C01805=1100.672,-5.062,-52.510,176.250,14.221,151.801
C01806=1100.666,-5.311,-52.497,176.248,14.221,151.801
C01807=1100.661,-5.561,-52.484,176.246,14.220,151.802
C01808=1100.655,-5.810,-52.470,176.244,14.220,151.802
C01809=1100.649,-6.060,-52.457,176.242,14.219,151.803
C01810=1100.643,-6.309,-52.443,176.240,14.219,151.803
C01811=1100.637,-6.559,-52.429,176.238,14.218,151.803
C01812=1100.631,-6.808,-52.416,176.236,14.218,151.804
C01813=1100.626,-7.058,-52.403,176.234,14.218,151.804
C01814=1100.620,-7.307,-52.390,176.232,14.217,151.804
C01815=1100.614,-7.557,-52.376,176.230,14.216,151.805
C01816=1100.608,-7.806,-52.363,176.228,14.216,151.805
C01817=1100.602,-8.055,-52.349,176.225,14.215,151.805
C01818=1100.597,-8.306,-52.336,176.223,14.214,151.806
C01819=1100.590,-8.555,-52.323,176.221,14.214,151.806
C01820=1100.585,-8.804,-52.309,176.219,14.213,151.807
C01821=1100.578,-9.054,-52.295,176.217,14.213,151.807
C01822=1100.573,-9.305,-52.282,176.215,14.212,151.807
C01823=1100.567,-9.554,-52.269,176.213,14.211,151.808
C01824=1100.561,-9.804,-52.255,176.210,14.211,151.808
C01825=1100.555,-10.053,-52.242,176.208,14.211,151.808
C01826=1100.550,-10.303,-52.229,176.206,14.210,151.809
C01827=1100.544,-10.552,-52.215,176.204,14.210,151.809
C01828=1100.537,-10.801,-52.202,176.202,14.209,151.809
C01829=1100.532,-11.052,-52.189,176.200,14.209,151.810
C01830=1100.526,-11.301,-52.176,176.198,14.208,151.810
C01831=1100.521,-11.551,-52.162,176.195,14.207,151.810
C01832=1100.515,-11.800,-52.149,176.193,14.206,151.811
C01833=1100.509,-12.050,-52.136,176.191,14.206,151.811
C01834=1100.503,-12.299,-52.122,176.189,14.205,151.811
C01835=1100.498,-12.548,-52.110,176.187,14.205,151.812
C01836=1100.492,-12.798,-52.096,176.185,14.204,151.812
C01837=1100.486,-13.047,-52.083,176.183,14.204,151.813
C01838=1100.480,-13.297,-52.070,176.181,14.203,151.813
C01839=1100.475,-13.547,-52.056,176.179,14.203,151.813
C01840=1100.468,-13.796,-52.043,176.177,14.202,151.813
C01841=1100.463,-14.046,-52.030,176.175,14.201,151.814
C01842=1100.457,-14.295,-52.017,176.173,14.201,151.814
C01843=1100.451,-14.545,-52.004,176.171,14.200,151.815
C01844=1100.446,-14.795,-51.990,176.169,14.200,151.815
C01845=1100.440,-15.045,-51.978,176.167,14.199,151.815
C01846=1100.434,-15.294,-51.965,176.165,14.198,151.816
C01847=1100.428,-15.544,-51.951,176.163,14.198,151.816
C01848=1100.422,-15.794,-51.938,176.160,14.197,151.816
C01849=1100.416,-16.061,-51.924,176.158,14.196,151.817
C01850=1100.409,-16.328,-51.910,176.156,14.196,151.817
C01851=1100.403,-16.596,-51.896,176.154,14.195,151.817
C01852=1100.397,-16.863,-51.882,176.152,14.195,151.818
C01853=1100.391,-17.113,-51.869,176.150,14.194,151.818
C01854=1100.385,-17.362,-51.856,176.148,14.194,151.818
C01855=1100.379,-17.612,-51.843,176.145,14.194,151.819
C01856=1100.373,-17.861,-51.830,176.144,14.193,151.819
C01857=1100.367,-18.111,-51.817,176.141,14.193,151.820
C01858=1100.362,-18.360,-51.804,176.140,14.192,151.820
C01859=1100.356,-18.610,-51.791,176.137,14.191,151.820
C01860=1100.350,-18.859,-51.778,176.135,14.190,151.821
C01861=1100.344,-19.109,-51.765,176.133,14.190,151.821
C01862=1100.338,-19.358,-51.752,176.131,14.189,151.821
C01863=1100.333,-19.609,-51.739,176.128,14.189,151.822
C01864=1100.327,-19.858,-51.726,176.127,14.188,151.822
C01865=1100.321,-20.108,-51.713,176.125,14.187,151.822
C01866=1100.315,-20.358,-51.701,176.123,14.187,151.823
C01867=1100.309,-20.607,-51.687,176.121,14.186,151.823
C01868=1100.303,-20.857,-51.675,176.118,14.186,151.823
C01869=1100.298,-21.106,-51.661,176.117,14.185,151.824
C01870=1100.292,-21.356,-51.649,176.114,14.185,151.824
C01871=1100.286,-21.606,-51.636,176.113,14.184,151.824
C01872=1100.280,-21.855,-51.623,176.110,14.184,151.825
C01873=1100.274,-22.105,-51.610,176.108,14.183,151.825
C01874=1100.268,-22.354,-51.597,176.106,14.183,151.825
C01875=1100.262,-22.604,-51.584,176.104,14.182,151.826
C01876=1100.257,-22.853,-51.572,176.102,14.181,151.826
C01877=1100.251,-23.103,-51.558,176.100,14.181,151.826
C01878=1100.245,-23.352,-51.546,176.098,14.180,151.827
C01879=1100.239,-23.602,-51.533,176.096,14.180,151.827
C01880=1100.233,-23.852,-51.520,176.094,14.179,151.827
C01881=1100.227,-24.101,-51.508,176.092,14.178,151.828
C01882=1100.221,-24.351,-51.495,176.090,14.178,151.828
C01883=1100.215,-24.600,-51.482,176.088,14.177,151.828
C01884=1100.210,-24.850,-51.469,176.086,14.177,151.829
C01885=1100.204,-25.100,-51.456,176.084,14.176,151.829
C01886=1100.198,-25.350,-51.444,176.082,14.176,151.829
C01887=1100.192,-25.599,-51.431,176.080,14.175,151.830
C01888=1100.187,-25.848,-51.418,176.078,14.174,151.830
C01889=1100.181,-26.098,-51.406,176.076,14.174,151.830
C01890=1100.175,-26.348,-51.393,176.074,14.173,151.831
C01891=1100.169,-26.597,-51.380,176.072,14.173,151.831
C01892=1100.163,-26.847,-51.367,176.070,14.172,151.831
C01893=1100.158,-27.096,-51.355,176.068,14.172,151.832
C01894=1100.152,-27.346,-51.343,176.066,14.171,151.832
C01895=1100.146,-27.596,-51.329,176.064,14.170,151.832
C01896=1100.140,-27.845,-51.317,176.062,14.170,151.833
C01897=1100.134,-28.095,-51.304,176.060,14.169,151.833
C01898=1100.128,-28.345,-51.292,176.058,14.169,151.833
C01899=1100.123,-28.594,-51.280,176.056,14.168,151.834
C01900=1100.116,-28.844,-51.266,176.054,14.168,151.834
C01901=1100.110,-29.094,-51.254,176.052,14.167,151.834
C01902=1100.105,-29.343,-51.241,176.050,14.166,151.835
C01903=1100.099,-29.593,-51.229,176.048,14.166,151.835
C01904=1100.093,-29.842,-51.216,176.046,14.165,151.835
C01905=1100.087,-30.092,-51.204,176.044,14.165,151.836
C01906=1100.080,-30.341,-51.191,176.042,14.164,151.836
C01907=1100.075,-30.591,-51.179,176.040,14.164,151.836
C01908=1100.069,-30.841,-51.166,176.038,14.163,151.837
C01909=1100.063,-31.090,-51.154,176.036,14.162,151.837
C01910=1100.057,-31.340,-51.141,176.034,14.162,151.837
C01911=1100.052,-31.590,-51.129,176.032,14.161,151.838
C01912=1100.046,-31.840,-51.116,176.030,14.161,151.838
C01913=1100.039,-32.106,-51.104,176.028,14.160,151.838
C01914=1100.033,-32.372,-51.089,176.026,14.160,151.839
C01915=1100.026,-32.639,-51.076,176.024,14.159,151.839
C01916=1100.021,-32.906,-51.063,176.022,14.158,151.839
C01917=1100.015,-33.156,-51.050,176.020,14.158,151.840
C01918=1100.008,-33.405,-51.038,176.018,14.157,151.840
C01919=1100.003,-33.654,-51.026,176.016,14.157,151.840
C01920=1099.997,-33.904,-51.014,176.014,14.156,151.841
C01921=1099.991,-34.154,-51.001,176.012,14.156,151.841
C01922=1099.985,-34.404,-50.989,176.010,14.155,151.841
C01923=1099.980,-34.653,-50.976,176.008,14.154,151.842
C01924=1099.973,-34.903,-50.964,176.006,14.154,151.842
C01925=1099.967,-35.153,-50.952,176.004,14.153,151.842
C01926=1099.962,-35.402,-50.940,176.002,14.153,151.843
C01927=1099.956,-35.652,-50.927,176.000,14.152,151.843
C01928=1099.950,-35.902,-50.915,175.998,14.152,151.843
C01929=1099.944,-36.152,-50.902,175.996,14.151,151.844
C01930=1099.938,-36.400,-50.890,175.994,14.151,151.844
C01931=1099.932,-36.650,-50.878,175.993,14.150,151.844
C01932=1099.927,-36.900,-50.865,175.991,14.150,151.844
C01933=1099.921,-37.149,-50.853,175.989,14.149,151.845
C01934=1099.915,-37.399,-50.841,175.987,14.148,151.845
C01935=1099.909,-37.649,-50.828,175.985,14.148,151.845
C01936=1099.903,-37.898,-50.816,175.983,14.147,151.846
C01937=1099.897,-38.148,-50.804,175.981,14.147,151.846
C01938=1099.892,-38.398,-50.791,175.978,14.146,151.847
C01939=1099.887,-38.648,-50.780,175.977,14.146,151.847
C01940=1099.880,-38.897,-50.768,175.975,14.145,151.847
C01941=1099.874,-39.147,-50.755,175.973,14.144,151.848
C01942=1099.869,-39.396,-50.743,175.971,14.144,151.848
C01943=1099.862,-39.646,-50.731,175.969,14.143,151.848
C01944=1099.856,-39.896,-50.719,175.967,14.143,151.848
C01945=1099.851,-40.145,-50.706,175.965,14.142,151.849
C01946=1099.844,-40.394,-50.694,175.963,14.142,151.849
C01947=1099.838,-40.644,-50.682,175.961,14.141,151.849
C01948=1099.833,-40.894,-50.670,175.959,14.141,151.850
C01949=1099.827,-41.144,-50.658,175.957,14.140,151.850
C01950=1099.821,-41.394,-50.646,175.956,14.140,151.850
C01951=1099.815,-41.643,-50.634,175.953,14.139,151.851
C01952=1099.809,-41.892,-50.622,175.951,14.139,151.851
C01953=1099.803,-42.142,-50.609,175.950,14.138,151.851
C01954=1099.797,-42.392,-50.598,175.947,14.137,151.852
C01955=1099.791,-42.642,-50.586,175.945,14.137,151.852
C01956=1099.785,-42.891,-50.573,175.943,14.136,151.852
C01957=1099.779,-43.140,-50.562,175.941,14.136,151.853
C01958=1099.773,-43.390,-50.549,175.940,14.135,151.853
C01959=1099.768,-43.641,-50.537,175.938,14.135,151.853
C01960=1099.762,-43.890,-50.526,175.936,14.134,151.854
C01961=1099.756,-44.139,-50.513,175.934,14.134,151.854
C01962=1099.750,-44.388,-50.502,175.932,14.133,151.854
C01963=1099.744,-44.639,-50.490,175.930,14.133,151.855
C01964=1099.738,-44.889,-50.477,175.928,14.132,151.855
C01965=1099.732,-45.138,-50.466,175.926,14.131,151.855
C01966=1099.726,-45.387,-50.453,175.924,14.131,151.856
C01967=1099.720,-45.638,-50.442,175.922,14.130,151.856
C01968=1099.715,-45.887,-50.430,175.920,14.130,151.856
C01969=1099.708,-46.136,-50.418,175.919,14.130,151.856
C01970=1099.703,-46.386,-50.406,175.917,14.129,151.857
C01971=1099.697,-46.636,-50.394,175.915,14.128,151.857
C01972=1099.691,-46.885,-50.382,175.913,14.128,151.858
C01973=1099.685,-47.135,-50.370,175.911,14.127,151.858
C01974=1099.679,-47.385,-50.358,175.909,14.127,151.858
C01975=1099.673,-47.634,-50.346,175.907,14.126,151.859
C01976=1099.667,-47.884,-50.335,175.905,14.126,151.859
C01977=1099.661,-48.151,-50.322,175.903,14.125,151.859
C01978=1099.655,-48.419,-50.309,175.901,14.124,151.859
C01979=1099.649,-48.685,-50.296,175.899,14.124,151.860
C01980=1099.643,-48.952,-50.284,175.897,14.123,151.860
C01981=1099.637,-49.202,-50.272,175.895,14.123,151.860
C01982=1099.630,-49.451,-50.260,175.893,14.122,151.861
C01983=1099.625,-49.701,-50.248,175.892,14.122,151.861
C01984=1099.618,-49.951,-50.236,175.890,14.121,151.861
C01985=1099.613,-50.200,-50.225,175.888,14.121,151.862
C01986=1099.607,-50.450,-50.213,175.886,14.120,151.862
C01987=1099.601,-50.699,-50.201,175.884,14.120,151.862
C01988=1099.595,-50.949,-50.189,175.882,14.119,151.863
C01989=1099.589,-51.198,-50.178,175.880,14.119,151.863
C01990=1099.583,-51.449,-50.166,175.878,14.118,151.863
C01991=1099.577,-51.698,-50.154,175.877,14.118,151.864
C01992=1099.571,-51.948,-50.143,175.875,14.117,151.864
C01993=1099.565,-52.198,-50.130,175.873,14.117,151.864
C01994=1099.559,-52.447,-50.119,175.871,14.116,151.865
C01995=1099.553,-52.697,-50.108,175.868,14.116,151.865
C01996=1099.546,-52.946,-50.096,175.867,14.115,151.865
C01997=1099.541,-53.196,-50.084,175.865,14.114,151.866
C01998=1099.534,-53.446,-50.072,175.863,14.115,151.866
C01999=1099.529,-53.695,-50.061,175.861,14.114,151.866
C02000=1099.523,-53.945,-50.049,175.859,14.114,151.867
C02001=1099.517,-54.195,-50.038,175.857,14.113,151.867
C02002=1099.510,-54.444,-50.026,175.855,14.112,151.867
C02003=1099.505,-54.694,-50.015,175.853,14.112,151.868
C02004=1099.499,-54.944,-50.003,175.851,14.111,151.868
C02005=1099.492,-55.194,-49.991,175.850,14.111,151.868
C02006=1099.486,-55.443,-49.980,175.848,14.111,151.869
C02007=1099.481,-55.693,-49.968,175.846,14.110,151.869
C02008=1099.475,-55.942,-49.956,175.844,14.110,151.869
C02009=1099.468,-56.192,-49.945,175.842,14.109,151.870
C02010=1099.462,-56.441,-49.933,175.840,14.109,151.870
C02011=1099.457,-56.692,-49.922,175.839,14.108,151.870
C02012=1099.451,-56.941,-49.911,175.837,14.108,151.870
C02013=1099.444,-57.191,-49.899,175.835,14.107,151.871
C02014=1099.439,-57.440,-49.888,175.833,14.107,151.871
C02015=1099.433,-57.690,-49.875,175.831,14.106,151.872
C02016=1099.427,-57.939,-49.864,175.829,14.106,151.872
C02017=1099.421,-58.190,-49.853,175.828,14.105,151.872
C02018=1099.415,-58.438,-49.842,175.825,14.105,151.872
C02019=1099.408,-58.689,-49.830,175.824,14.104,151.873
C02020=1099.403,-58.938,-49.818,175.821,14.104,151.873
C02021=1099.397,-59.188,-49.807,175.820,14.103,151.873
C02022=1099.391,-59.438,-49.796,175.818,14.103,151.874
C02023=1099.384,-59.687,-49.784,175.816,14.103,151.874
C02024=1099.379,-59.937,-49.773,175.814,14.102,151.874
C02025=1099.373,-60.187,-49.761,175.812,14.102,151.875
C02026=1099.367,-60.436,-49.750,175.810,14.101,151.875
C02027=1099.361,-60.685,-49.739,175.808,14.100,151.875
C02028=1099.355,-60.936,-49.728,175.807,14.101,151.876
C02029=1099.349,-61.185,-49.716,175.805,14.100,151.876
C02030=1099.343,-61.435,-49.704,175.803,14.099,151.876
C02031=1099.337,-61.685,-49.693,175.801,14.099,151.877
C02032=1099.331,-61.934,-49.681,175.799,14.098,151.877
C02033=1099.325,-62.184,-49.671,175.798,14.098,151.877
C02034=1099.319,-62.434,-49.659,175.796,14.098,151.878
C02035=1099.314,-62.684,-49.648,175.794,14.097,151.878
C02036=1099.308,-62.932,-49.636,175.792,14.097,151.878
C02037=1099.301,-63.183,-49.625,175.790,14.096,151.879
C02038=1099.296,-63.432,-49.614,175.788,14.095,151.879
C02039=1099.289,-63.682,-49.603,175.787,14.095,151.879
C02040=1099.283,-63.931,-49.591,175.785,14.095,151.879
C02041=1099.278,-64.200,-49.579,175.783,14.094,151.880
C02042=1099.271,-64.468,-49.567,175.781,14.094,151.880
C02043=1099.264,-64.736,-49.554,175.778,14.093,151.881
C02044=1099.258,-65.005,-49.543,175.777,14.093,151.881
C02045=1099.252,-65.254,-49.532,175.775,14.092,151.881
C02046=1099.246,-65.504,-49.521,175.773,14.092,151.882
C02047=1099.240,-65.754,-49.510,175.771,14.091,151.882
C02048=1099.235,-66.003,-49.498,175.769,14.091,151.882
C02049=1099.228,-66.253,-49.486,175.767,14.090,151.883
C02050=1099.223,-66.503,-49.475,175.765,14.090,151.883
C02051=1099.217,-66.752,-49.465,175.764,14.090,151.883
C02052=1099.210,-67.002,-49.453,175.762,14.089,151.883
C02053=1099.205,-67.252,-49.442,175.760,14.088,151.884
C02054=1099.198,-67.501,-49.430,175.758,14.088,151.884
C02055=1099.192,-67.751,-49.420,175.757,14.088,151.884
C02056=1099.187,-68.000,-49.409,175.755,14.088,151.885
C02057=1099.181,-68.251,-49.397,175.753,14.087,151.885
C02058=1099.175,-68.500,-49.386,175.751,14.086,151.885
C02059=1099.170,-68.750,-49.375,175.749,14.086,151.886
C02060=1099.163,-69.000,-49.364,175.748,14.086,151.886
C02061=1099.157,-69.250,-49.353,175.746,14.085,151.886
C02062=1099.152,-69.499,-49.342,175.744,14.085,151.887
C02063=1099.145,-69.749,-49.330,175.742,14.084,151.887
C02064=1099.139,-69.998,-49.319,175.741,14.084,151.887
C02065=1099.134,-70.248,-49.308,175.738,14.083,151.888
C02066=1099.128,-70.497,-49.298,175.737,14.083,151.888
C02067=1099.121,-70.747,-49.286,175.734,14.082,151.888
C02068=1099.116,-70.997,-49.275,175.733,14.082,151.889
C02069=1099.110,-71.246,-49.265,175.731,14.081,151.889
C02070=1099.104,-71.496,-49.253,175.729,14.081,151.889
C02071=1099.098,-71.746,-49.242,175.727,14.080,151.889
C02072=1099.093,-71.996,-49.231,175.725,14.080,151.890
C02073=1099.087,-72.245,-49.220,175.724,14.080,151.890
C02074=1099.081,-72.495,-49.209,175.722,14.079,151.890
C02075=1099.075,-72.745,-49.198,175.720,14.078,151.891
C02076=1099.069,-72.994,-49.187,175.718,14.078,151.891
C02077=1099.063,-73.245,-49.176,175.717,14.078,151.891
C02078=1099.057,-73.494,-49.165,175.715,14.077,151.892
C02079=1099.052,-73.744,-49.154,175.713,14.077,151.892
C02080=1099.046,-73.993,-49.143,175.711,14.076,151.892
C02081=1099.039,-74.243,-49.132,175.710,14.077,151.893
C02082=1099.034,-74.493,-49.121,175.708,14.076,151.893
C02083=1099.028,-74.742,-49.110,175.706,14.075,151.893
C02084=1099.022,-74.991,-49.100,175.704,14.075,151.894
C02085=1099.015,-75.242,-49.089,175.703,14.075,151.894
C02086=1099.009,-75.491,-49.078,175.700,14.074,151.894
C02087=1099.004,-75.741,-49.067,175.698,14.074,151.895
C02088=1098.997,-75.991,-49.056,175.697,14.074,151.895
C02089=1098.992,-76.240,-49.045,175.695,14.073,151.895
C02090=1098.986,-76.490,-49.034,175.693,14.072,151.896
C02091=1098.979,-76.740,-49.023,175.691,14.072,151.896
C02092=1098.973,-76.990,-49.013,175.690,14.072,151.896
C02093=1098.968,-77.239,-49.002,175.688,14.072,151.897
C02094=1098.962,-77.489,-48.991,175.686,14.071,151.897
C02095=1098.956,-77.739,-48.980,175.685,14.071,151.897
C02096=1098.950,-77.988,-48.969,175.683,14.071,151.898
C02097=1098.943,-78.238,-48.959,175.681,14.070,151.898
C02098=1098.938,-78.487,-48.948,175.678,14.070,151.898
C02099=1098.931,-78.737,-48.937,175.677,14.069,151.898
C02100=1098.926,-78.987,-48.926,175.675,14.069,151.899
C02101=1098.920,-79.237,-48.916,175.673,14.068,151.899
C02102=1098.914,-79.486,-48.905,175.672,14.068,151.899
C02103=1098.907,-79.736,-48.894,175.670,14.068,151.900
C02104=1098.902,-79.986,-48.883,175.668,14.067,151.900
C02105=1098.895,-80.256,-48.871,175.666,14.067,151.901
C02106=1098.889,-80.527,-48.860,175.664,14.066,151.901
C02107=1098.882,-80.797,-48.849,175.663,14.066,151.901
C02108=1098.875,-81.068,-48.837,175.660,14.066,151.902
C02109=1098.870,-81.318,-48.826,175.658,14.065,151.902
C02110=1098.863,-81.567,-48.816,175.656,14.065,151.902
C02111=1098.857,-81.817,-48.805,175.655,14.065,151.903
C02112=1098.851,-82.066,-48.794,175.653,14.065,151.903
C02113=1098.845,-82.316,-48.784,175.651,14.064,151.903
C02114=1098.839,-82.566,-48.773,175.650,14.064,151.904
C02115=1098.832,-82.816,-48.763,175.648,14.064,151.904
C02116=1098.826,-83.065,-48.752,175.646,14.063,151.904
C02117=1098.821,-83.315,-48.742,175.644,14.063,151.905
C02118=1098.814,-83.564,-48.731,175.643,14.062,151.905
C02119=1098.808,-83.815,-48.720,175.640,14.062,151.905
C02120=1098.802,-84.064,-48.709,175.639,14.062,151.906
C02121=1098.796,-84.314,-48.700,175.637,14.062,151.906
C02122=1098.790,-84.563,-48.689,175.635,14.061,151.906
C02123=1098.784,-84.814,-48.678,175.634,14.061,151.907
C02124=1098.778,-85.063,-48.667,175.632,14.061,151.907
C02125=1098.772,-85.313,-48.657,175.630,14.060,151.907
C02126=1098.766,-85.562,-48.647,175.629,14.060,151.908
C02127=1098.760,-85.811,-48.636,175.626,14.060,151.908
C02128=1098.754,-86.062,-48.625,175.625,14.059,151.908
C02129=1098.748,-86.311,-48.615,175.623,14.059,151.909
C02130=1098.742,-86.561,-48.604,175.621,14.059,151.909
C02131=1098.735,-86.810,-48.594,175.619,14.058,151.909
C02132=1098.730,-87.060,-48.584,175.618,14.058,151.910
C02133=1098.724,-87.310,-48.573,175.616,14.058,151.910
C02134=1098.717,-87.560,-48.562,175.614,14.057,151.910
C02135=1098.712,-87.810,-48.552,175.612,14.058,151.911
C02136=1098.705,-88.059,-48.542,175.610,14.057,151.911
C02137=1098.699,-88.308,-48.531,175.608,14.057,151.911
C02138=1098.693,-88.559,-48.520,175.607,14.056,151.912
C02139=1098.687,-88.808,-48.510,175.605,14.056,151.912
C02140=1098.681,-89.058,-48.500,175.603,14.055,151.912
C02141=1098.675,-89.308,-48.490,175.602,14.056,151.913
C02142=1098.669,-89.557,-48.479,175.600,14.055,151.913
C02143=1098.663,-89.807,-48.469,175.598,14.055,151.913
C02144=1098.657,-90.056,-48.458,175.596,14.055,151.914
C02145=1098.651,-90.307,-48.448,175.594,14.054,151.914
C02146=1098.645,-90.556,-48.438,175.593,14.054,151.914
C02147=1098.639,-90.806,-48.427,175.591,14.054,151.915
C02148=1098.633,-91.056,-48.417,175.589,14.053,151.915
C02149=1098.627,-91.305,-48.406,175.588,14.053,151.915
C02150=1098.621,-91.555,-48.397,175.586,14.053,151.916
C02151=1098.615,-91.804,-48.386,175.584,14.052,151.916
C02152=1098.608,-92.055,-48.376,175.582,14.052,151.916
C02153=1098.603,-92.304,-48.365,175.580,14.052,151.917
C02154=1098.596,-92.554,-48.355,175.578,14.051,151.917
C02155=1098.591,-92.804,-48.345,175.577,14.052,151.917
C02156=1098.584,-93.053,-48.334,175.575,14.051,151.918
C02157=1098.579,-93.303,-48.324,175.574,14.051,151.918
C02158=1098.573,-93.553,-48.313,175.572,14.050,151.918
C02159=1098.567,-93.802,-48.304,175.570,14.050,151.919
C02160=1098.561,-94.052,-48.293,175.568,14.050,151.919
C02161=1098.554,-94.302,-48.283,175.566,14.050,151.919
C02162=1098.549,-94.552,-48.272,175.564,14.049,151.920
C02163=1098.543,-94.802,-48.262,175.563,14.049,151.920
C02164=1098.537,-95.051,-48.252,175.561,14.049,151.920
C02165=1098.531,-95.301,-48.242,175.560,14.049,151.921
C02166=1098.525,-95.550,-48.231,175.558,14.048,151.921
C02167=1098.519,-95.800,-48.222,175.555,14.048,151.921
C02168=1098.513,-96.050,-48.211,175.554,14.048,151.922
C02169=1098.506,-96.323,-48.201,175.552,14.048,151.922
C02170=1098.500,-96.595,-48.189,175.550,14.047,151.922
C02171=1098.493,-96.868,-48.178,175.549,14.047,151.923
C02172=1098.486,-97.141,-48.167,175.547,14.047,151.923
C02173=1098.481,-97.391,-48.156,175.545,14.046,151.923
C02174=1098.474,-97.640,-48.146,175.543,14.046,151.924
C02175=1098.469,-97.890,-48.136,175.541,14.046,151.924
C02176=1098.463,-98.140,-48.126,175.539,14.045,151.925
C02177=1098.456,-98.389,-48.116,175.538,14.045,151.925
C02178=1098.451,-98.640,-48.106,175.536,14.045,151.925
C02179=1098.444,-98.889,-48.096,175.535,14.045,151.926
C02180=1098.438,-99.138,-48.086,175.533,14.045,151.926
C02181=1098.433,-99.389,-48.076,175.530,14.044,151.926
C02182=1098.426,-99.638,-48.066,175.529,14.044,151.927
C02183=1098.420,-99.888,-48.056,175.527,14.044,151.927
C02184=1098.413,-100.137,-48.045,175.526,14.044,151.927
C02185=1098.408,-100.388,-48.035,175.524,14.044,151.928
C02186=1098.401,-100.637,-48.026,175.522,14.044,151.928
C02187=1098.395,-100.887,-48.015,175.520,14.043,151.928
C02188=1098.389,-101.137,-48.005,175.518,14.043,151.929
C02189=1098.383,-101.386,-47.996,175.517,14.043,151.929
C02190=1098.377,-101.636,-47.985,175.515,14.042,151.929
C02191=1098.371,-101.886,-47.975,175.514,14.043,151.930
C02192=1098.365,-102.136,-47.966,175.512,14.042,151.930
C02193=1098.359,-102.385,-47.955,175.510,14.042,151.931
C02194=1098.353,-102.634,-47.946,175.508,14.042,151.931
C02195=1098.347,-102.885,-47.936,175.506,14.041,151.931
C02196=1098.341,-103.134,-47.925,175.505,14.041,151.931
C02197=1098.334,-103.384,-47.916,175.503,14.041,151.932
C02198=1098.329,-103.634,-47.906,175.501,14.041,151.932
C02199=1098.323,-103.883,-47.896,175.499,14.041,151.933
C02200=1098.316,-104.133,-47.886,175.498,14.041,151.933
C02201=1098.310,-104.382,-47.876,175.496,14.040,151.933
C02202=1098.305,-104.633,-47.866,175.495,14.041,151.934
C02203=1098.298,-104.882,-47.856,175.493,14.040,151.934
C02204=1098.292,-105.132,-47.846,175.491,14.040,151.934
C02205=1098.286,-105.381,-47.837,175.489,14.040,151.935
C02206=1098.280,-105.631,-47.827,175.487,14.039,151.935
C02207=1098.274,-105.881,-47.816,175.486,14.039,151.935
C02208=1098.268,-106.130,-47.807,175.484,14.039,151.936
C02209=1098.262,-106.380,-47.797,175.483,14.039,151.936
C02210=1098.256,-106.630,-47.788,175.480,14.039,151.936
C02211=1098.250,-106.880,-47.777,175.479,14.039,151.937
C02212=1098.244,-107.129,-47.767,175.477,14.038,151.937
C02213=1098.237,-107.379,-47.758,175.476,14.039,151.938
C02214=1098.231,-107.629,-47.748,175.474,14.038,151.938
C02215=1098.225,-107.879,-47.738,175.472,14.038,151.938
C02216=1098.219,-108.129,-47.729,175.470,14.038,151.939
C02217=1098.213,-108.378,-47.718,175.468,14.037,151.939
C02218=1098.207,-108.628,-47.708,175.467,14.038,151.939
C02219=1098.201,-108.878,-47.699,175.465,14.037,151.940
C02220=1098.195,-109.127,-47.689,175.463,14.037,151.940
C02221=1098.189,-109.377,-47.680,175.461,14.037,151.940
C02222=1098.182,-109.627,-47.670,175.460,14.037,151.941
C02223=1098.176,-109.876,-47.660,175.458,14.037,151.941
C02224=1098.170,-110.126,-47.650,175.456,14.037,151.941
C02225=1098.164,-110.376,-47.641,175.455,14.036,151.942
C02226=1098.158,-110.626,-47.631,175.453,14.037,151.942
C02227=1098.152,-110.876,-47.621,175.451,14.036,151.943
C02228=1098.146,-111.125,-47.611,175.450,14.036,151.943
C02229=1098.140,-111.375,-47.602,175.448,14.036,151.943
C02230=1098.133,-111.624,-47.592,175.446,14.036,151.944
C02231=1098.127,-111.874,-47.582,175.444,14.036,151.944
C02232=1098.121,-112.124,-47.572,175.443,14.036,151.944
C02233=1098.115,-112.363,-47.563,175.441,14.036,151.945
C02234=1098.109,-112.602,-47.554,175.440,14.036,151.945
C02235=1098.103,-112.841,-47.545,175.437,14.035,151.945
C02236=1098.098,-113.081,-47.536,175.436,14.036,151.946
C02237=1098.091,-113.319,-47.526,175.434,14.035,151.946
C02238=1098.085,-113.559,-47.517,175.433,14.035,151.946
C02239=1098.080,-113.798,-47.507,175.431,14.035,151.947
C02240=1098.073,-114.037,-47.499,175.429,14.035,151.947
C02241=1098.067,-114.287,-47.489,175.428,14.035,151.948
C02242=1098.062,-114.536,-47.480,175.426,14.034,151.948
C02243=1098.056,-114.786,-47.470,175.425,14.035,151.948
C02244=1098.049,-115.036,-47.461,175.422,14.035,151.949
C02245=1098.043,-115.285,-47.451,175.421,14.034,151.949
C02246=1098.037,-115.535,-47.442,175.419,14.034,151.949
C02247=1098.031,-115.785,-47.432,175.418,14.035,151.950
C02248=1098.025,-116.035,-47.422,175.415,14.034,151.950
C02249=1098.019,-116.285,-47.413,175.414,14.034,151.950
C02250=1098.012,-116.534,-47.403,175.412,14.034,151.951
C02251=1098.006,-116.784,-47.394,175.411,14.034,151.951
C02252=1098.000,-117.034,-47.384,175.409,14.033,151.951
C02253=1097.994,-117.284,-47.375,175.407,14.034,151.952
C02254=1097.988,-117.534,-47.365,175.405,14.034,151.952
C02255=1097.981,-117.783,-47.355,175.404,14.034,151.953
C02256=1097.975,-118.033,-47.346,175.402,14.033,151.953
C02257=1097.970,-118.282,-47.337,175.400,14.034,151.953
C02258=1097.964,-118.532,-47.327,175.398,14.033,151.954
C02259=1097.957,-118.782,-47.318,175.397,14.033,151.954
C02260=1097.951,-119.032,-47.308,175.395,14.033,151.954
C02261=1097.945,-119.281,-47.298,175.393,14.033,151.955
C02262=1097.939,-119.531,-47.289,175.392,14.034,151.955
C02263=1097.933,-119.781,-47.279,175.390,14.033,151.956
C02264=1097.926,-120.030,-47.270,175.389,14.033,151.956
C02265=1097.920,-120.280,-47.261,175.386,14.033,151.956
C02266=1097.914,-120.531,-47.252,175.385,14.033,151.957
C02267=1097.908,-120.781,-47.242,175.383,14.033,151.957
C02268=1097.902,-121.030,-47.233,175.382,14.033,151.957
C02269=1097.896,-121.279,-47.224,175.379,14.033,151.958
C02270=1097.890,-121.529,-47.214,175.378,14.033,151.958
C02271=1097.884,-121.779,-47.204,175.376,14.032,151.959
C02272=1097.877,-122.029,-47.195,175.375,14.033,151.959
C02273=1097.870,-122.278,-47.186,175.373,14.033,151.959
C02274=1097.864,-122.528,-47.176,175.371,14.033,151.960
C02275=1097.858,-122.778,-47.167,175.370,14.033,151.960
C02276=1097.853,-123.028,-47.158,175.368,14.032,151.960
C02277=1097.847,-123.277,-47.149,175.366,14.033,151.961
C02278=1097.840,-123.527,-47.139,175.364,14.032,151.961
C02279=1097.834,-123.777,-47.130,175.363,14.033,151.962
C02280=1097.827,-124.026,-47.121,175.361,14.032,151.962
C02281=1097.821,-124.276,-47.111,175.359,14.032,151.962
C02282=1097.815,-124.527,-47.102,175.358,14.033,151.963
C02283=1097.810,-124.776,-47.093,175.356,14.033,151.963
C02284=1097.804,-125.026,-47.083,175.354,14.032,151.963
C02285=1097.797,-125.275,-47.074,175.352,14.032,151.964
C02286=1097.791,-125.525,-47.065,175.351,14.033,151.964
C02287=1097.784,-125.775,-47.055,175.349,14.032,151.965
C02288=1097.779,-126.025,-47.046,175.347,14.033,151.965
C02289=1097.772,-126.275,-47.037,175.346,14.033,151.965
C02290=1097.765,-126.524,-47.028,175.344,14.032,151.966
C02291=1097.760,-126.773,-47.019,175.342,14.033,151.966
C02292=1097.754,-127.024,-47.010,175.340,14.032,151.967
C02293=1097.746,-127.319,-46.999,175.339,14.033,151.967
C02294=1097.739,-127.615,-46.987,175.337,14.032,151.967
C02295=1097.731,-127.911,-46.977,175.334,14.032,151.968
C02296=1097.726,-128.206,-46.966,175.333,14.033,151.968
C02297=1097.317,-128.228,-47.072,175.291,14.129,151.996
C02298=1097.321,-127.958,-47.082,175.293,14.130,151.996
C02299=1097.328,-127.689,-47.092,175.295,14.129,151.996
C02300=1097.335,-127.419,-47.102,175.297,14.130,151.995
C02301=1097.341,-127.150,-47.112,175.298,14.129,151.995
C02302=1097.347,-126.900,-47.121,175.300,14.130,151.995
C02303=1097.353,-126.650,-47.130,175.302,14.130,151.994
C02304=1097.359,-126.400,-47.140,175.304,14.130,151.994
C02305=1097.366,-126.151,-47.149,175.305,14.129,151.993
C02306=1097.372,-125.901,-47.158,175.307,14.129,151.993
C02307=1097.378,-125.652,-47.167,175.308,14.130,151.993
C02308=1097.384,-125.401,-47.176,175.310,14.129,151.992
C02309=1097.391,-125.152,-47.185,175.312,14.130,151.992
C02310=1097.397,-124.902,-47.195,175.314,14.129,151.991
C02311=1097.403,-124.652,-47.204,175.315,14.130,151.991
C02312=1097.409,-124.402,-47.214,175.317,14.130,151.991
C02313=1097.415,-124.152,-47.223,175.318,14.129,151.990
C02314=1097.421,-123.903,-47.231,175.321,14.130,151.990
C02315=1097.427,-123.653,-47.241,175.322,14.130,151.990
C02316=1097.434,-123.404,-47.250,175.324,14.130,151.989
C02317=1097.440,-123.154,-47.260,175.325,14.130,151.989
C02318=1097.446,-122.904,-47.270,175.327,14.130,151.989
C02319=1097.452,-122.654,-47.279,175.329,14.130,151.988
C02320=1097.458,-122.404,-47.288,175.331,14.130,151.988
C02321=1097.464,-122.155,-47.297,175.332,14.130,151.987
C02322=1097.470,-121.905,-47.306,175.334,14.131,151.987
C02323=1097.477,-121.655,-47.316,175.336,14.130,151.987
C02324=1097.483,-121.406,-47.325,175.337,14.130,151.986
C02325=1097.489,-121.156,-47.335,175.339,14.131,151.986
C02326=1097.495,-120.906,-47.344,175.340,14.130,151.986
C02327=1097.501,-120.656,-47.354,175.343,14.130,151.985
C02328=1097.508,-120.406,-47.364,175.344,14.130,151.985
C02329=1097.513,-120.156,-47.372,175.346,14.131,151.984
C02330=1097.520,-119.907,-47.381,175.347,14.131,151.984
C02331=1097.526,-119.657,-47.391,175.350,14.131,151.984
C02332=1097.532,-119.408,-47.400,175.351,14.131,151.983
C02333=1097.538,-119.158,-47.410,175.353,14.131,151.983
C02334=1097.544,-118.908,-47.419,175.354,14.131,151.983
C02335=1097.551,-118.658,-47.429,175.356,14.132,151.982
C02336=1097.557,-118.408,-47.438,175.358,14.131,151.982
C02337=1097.563,-118.159,-47.448,175.360,14.131,151.981
C02338=1097.569,-117.909,-47.458,175.361,14.132,151.981
C02339=1097.575,-117.659,-47.467,175.363,14.132,151.981
C02340=1097.581,-117.409,-47.477,175.365,14.131,151.980
C02341=1097.587,-117.160,-47.486,175.366,14.132,151.980
C02342=1097.593,-116.910,-47.496,175.368,14.132,151.980
C02343=1097.599,-116.661,-47.505,175.370,14.132,151.979
C02344=1097.605,-116.411,-47.515,175.371,14.132,151.979
C02345=1097.612,-116.161,-47.524,175.373,14.132,151.979
C02346=1097.618,-115.911,-47.534,175.375,14.132,151.978
C02347=1097.624,-115.661,-47.543,175.377,14.133,151.978
C02348=1097.630,-115.412,-47.553,175.378,14.132,151.978
C02349=1097.636,-115.162,-47.562,175.380,14.133,151.977
C02350=1097.643,-114.912,-47.572,175.382,14.133,151.977
C02351=1097.649,-114.662,-47.582,175.384,14.133,151.977
C02352=1097.655,-114.412,-47.591,175.385,14.133,151.976
C02353=1097.661,-114.163,-47.601,175.387,14.133,151.976
C02354=1097.667,-113.913,-47.610,175.388,14.133,151.975
C02355=1097.673,-113.663,-47.620,175.391,14.133,151.975
C02356=1097.679,-113.414,-47.629,175.392,14.133,151.975
C02357=1097.685,-113.164,-47.639,175.394,14.134,151.974
C02358=1097.691,-112.909,-47.649,175.395,14.133,151.974
C02359=1097.698,-112.654,-47.658,175.397,14.134,151.974
C02360=1097.704,-112.399,-47.668,175.399,14.134,151.973
C02361=1097.710,-112.145,-47.678,175.401,14.135,151.973
C02362=1097.716,-111.895,-47.688,175.402,14.134,151.973
C02363=1097.723,-111.646,-47.698,175.404,14.134,151.972
C02364=1097.729,-111.396,-47.707,175.405,14.135,151.972
C02365=1097.735,-111.146,-47.717,175.408,14.135,151.972
C02366=1097.741,-110.896,-47.727,175.409,14.134,151.971
C02367=1097.747,-110.646,-47.736,175.411,14.135,151.971
C02368=1097.753,-110.397,-47.746,175.412,14.135,151.970
C02369=1097.760,-110.147,-47.755,175.414,14.136,151.970
C02370=1097.765,-109.897,-47.766,175.416,14.135,151.970
C02371=1097.772,-109.647,-47.776,175.418,14.135,151.969
C02372=1097.778,-109.398,-47.785,175.420,14.136,151.969
C02373=1097.784,-109.148,-47.795,175.421,14.136,151.969
C02374=1097.790,-108.898,-47.804,175.423,14.137,151.968
C02375=1097.796,-108.648,-47.814,175.425,14.136,151.968
C02376=1097.803,-108.399,-47.824,175.427,14.136,151.968
C02377=1097.809,-108.149,-47.834,175.428,14.137,151.967
C02378=1097.815,-107.900,-47.843,175.430,14.137,151.967
C02379=1097.820,-107.649,-47.854,175.431,14.137,151.967
C02380=1097.827,-107.400,-47.863,175.433,14.137,151.966
C02381=1097.833,-107.150,-47.873,175.435,14.137,151.966
C02382=1097.839,-106.901,-47.883,175.437,14.138,151.966
C02383=1097.845,-106.651,-47.893,175.438,14.137,151.965
C02384=1097.851,-106.401,-47.903,175.440,14.138,151.965
C02385=1097.857,-106.151,-47.912,175.442,14.138,151.965
C02386=1097.864,-105.902,-47.923,175.443,14.138,151.964
C02387=1097.870,-105.652,-47.932,175.446,14.139,151.964
C02388=1097.876,-105.402,-47.942,175.447,14.139,151.964
C02389=1097.881,-105.152,-47.952,175.449,14.139,151.963
C02390=1097.888,-104.903,-47.962,175.450,14.139,151.963
C02391=1097.894,-104.653,-47.972,175.452,14.139,151.963
C02392=1097.900,-104.403,-47.981,175.454,14.139,151.962
C02393=1097.906,-104.153,-47.991,175.455,14.140,151.962
C02394=1097.912,-103.904,-48.002,175.458,14.140,151.961
C02395=1097.918,-103.654,-48.011,175.459,14.140,151.961
C02396=1097.924,-103.404,-48.021,175.461,14.140,151.961
C02397=1097.930,-103.154,-48.031,175.462,14.141,151.961
C02398=1097.936,-102.905,-48.041,175.464,14.141,151.960
C02399=1097.942,-102.655,-48.051,175.465,14.141,151.960
C02400=1097.949,-102.404,-48.061,175.468,14.141,151.959
C02401=1097.955,-102.155,-48.072,175.470,14.142,151.959
C02402=1097.961,-101.906,-48.081,175.471,14.142,151.959
C02403=1097.967,-101.656,-48.091,175.473,14.142,151.958
C02404=1097.973,-101.406,-48.102,175.474,14.142,151.958
C02405=1097.979,-101.156,-48.111,175.476,14.142,151.958
C02406=1097.985,-100.907,-48.121,175.478,14.143,151.957
C02407=1097.991,-100.657,-48.132,175.480,14.143,151.957
C02408=1097.997,-100.407,-48.141,175.482,14.143,151.957
C02409=1098.003,-100.158,-48.151,175.483,14.143,151.956
C02410=1098.009,-99.908,-48.162,175.485,14.144,151.956
C02411=1098.015,-99.658,-48.171,175.486,14.143,151.956
C02412=1098.022,-99.408,-48.181,175.488,14.144,151.955
C02413=1098.027,-99.159,-48.192,175.490,14.145,151.955
C02414=1098.033,-98.909,-48.201,175.492,14.145,151.955
C02415=1098.041,-98.659,-48.212,175.494,14.145,151.954
C02416=1098.047,-98.409,-48.221,175.495,14.145,151.954
C02417=1098.052,-98.159,-48.232,175.497,14.145,151.954
C02418=1098.059,-97.910,-48.242,175.499,14.146,151.953
C02419=1098.064,-97.660,-48.252,175.500,14.146,151.953
C02420=1098.071,-97.411,-48.262,175.502,14.146,151.953
C02421=1098.077,-97.161,-48.272,175.504,14.146,151.952
C02422=1098.083,-96.889,-48.283,175.506,14.147,151.952
C02423=1098.090,-96.616,-48.294,175.508,14.147,151.952
C02424=1098.096,-96.342,-48.305,175.510,14.147,151.951
C02425=1098.103,-96.069,-48.317,175.512,14.148,151.951
C02426=1098.109,-95.820,-48.328,175.513,14.148,151.951
C02427=1098.115,-95.570,-48.337,175.515,14.148,151.950
C02428=1098.120,-95.320,-48.347,175.517,14.148,151.950
C02429=1098.127,-95.071,-48.358,175.519,14.149,151.950
C02430=1098.132,-94.821,-48.368,175.520,14.150,151.949
C02431=1098.139,-94.572,-48.378,175.522,14.149,151.949
C02432=1098.144,-94.321,-48.388,175.524,14.150,151.949
C02433=1098.151,-94.072,-48.399,175.526,14.150,151.948
C02434=1098.156,-93.821,-48.409,175.527,14.150,151.948
C02435=1098.163,-93.572,-48.419,175.529,14.151,151.948
C02436=1098.168,-93.322,-48.429,175.530,14.151,151.947
C02437=1098.175,-93.073,-48.440,175.533,14.151,151.947
C02438=1098.180,-92.823,-48.450,175.534,14.152,151.947
C02439=1098.187,-92.574,-48.460,175.536,14.152,151.946
C02440=1098.192,-92.324,-48.470,175.538,14.152,151.946
C02441=1098.199,-92.074,-48.481,175.540,14.153,151.946
C02442=1098.204,-91.825,-48.491,175.541,14.153,151.945
C02443=1098.210,-91.574,-48.502,175.543,14.153,151.945
C02444=1098.217,-91.325,-48.512,175.545,14.154,151.945
C02445=1098.222,-91.075,-48.522,175.546,14.154,151.944
C02446=1098.229,-90.826,-48.533,175.548,14.155,151.944
C02447=1098.234,-90.576,-48.543,175.550,14.154,151.944
C02448=1098.241,-90.326,-48.553,175.551,14.155,151.943
C02449=1098.247,-90.077,-48.564,175.554,14.155,151.943
C02450=1098.253,-89.826,-48.574,175.555,14.155,151.943
C02451=1098.259,-89.577,-48.585,175.557,14.156,151.942
C02452=1098.264,-89.327,-48.595,175.559,14.156,151.942
C02453=1098.271,-89.078,-48.605,175.560,14.156,151.942
C02454=1098.277,-88.828,-48.616,175.562,14.157,151.941
C02455=1098.283,-88.578,-48.626,175.564,14.158,151.941
C02456=1098.289,-88.328,-48.637,175.565,14.157,151.941
C02457=1098.296,-88.079,-48.647,175.567,14.158,151.940
C02458=1098.301,-87.829,-48.657,175.570,14.158,151.940
C02459=1098.307,-87.579,-48.668,175.571,14.158,151.940
C02460=1098.313,-87.330,-48.678,175.573,14.159,151.939
C02461=1098.319,-87.080,-48.689,175.575,14.159,151.939
C02462=1098.326,-86.830,-48.699,175.576,14.159,151.939
C02463=1098.331,-86.580,-48.710,175.578,14.160,151.938
C02464=1098.337,-86.331,-48.720,175.580,14.160,151.938
C02465=1098.343,-86.081,-48.731,175.581,14.160,151.938
C02466=1098.350,-85.831,-48.742,175.583,14.161,151.938
C02467=1098.356,-85.581,-48.751,175.585,14.161,151.937
C02468=1098.362,-85.332,-48.762,175.587,14.161,151.937
C02469=1098.367,-85.082,-48.773,175.588,14.162,151.937
C02470=1098.374,-84.833,-48.783,175.591,14.162,151.936
C02471=1098.380,-84.582,-48.794,175.592,14.162,151.936
C02472=1098.386,-84.333,-48.804,175.594,14.163,151.936
C02473=1098.392,-84.084,-48.815,175.596,14.163,151.935
C02474=1098.398,-83.834,-48.825,175.597,14.164,151.935
C02475=1098.405,-83.584,-48.836,175.599,14.164,151.935
C02476=1098.410,-83.334,-48.847,175.601,14.165,151.934
C02477=1098.416,-83.085,-48.858,175.603,14.165,151.934
C02478=1098.422,-82.835,-48.867,175.604,14.165,151.934
C02479=1098.429,-82.585,-48.879,175.607,14.165,151.933
C02480=1098.434,-82.335,-48.889,175.608,14.166,151.933
C02481=1098.441,-82.086,-48.900,175.610,14.166,151.933
C02482=1098.447,-81.837,-48.911,175.612,14.166,151.932
C02483=1098.453,-81.586,-48.921,175.614,14.167,151.932
C02484=1098.459,-81.337,-48.931,175.615,14.167,151.932
C02485=1098.465,-81.087,-48.942,175.617,14.168,151.931
C02486=1098.472,-80.817,-48.954,175.619,14.168,151.931
C02487=1098.478,-80.546,-48.966,175.621,14.169,151.931
C02488=1098.485,-80.275,-48.977,175.623,14.169,151.930
C02489=1098.491,-80.005,-48.989,175.625,14.170,151.930
C02490=1098.497,-79.755,-49.000,175.627,14.169,151.930
C02491=1098.504,-79.505,-49.010,175.628,14.170,151.929
C02492=1098.510,-79.256,-49.021,175.630,14.171,151.929
C02493=1098.515,-79.006,-49.031,175.632,14.170,151.929
C02494=1098.521,-78.756,-49.042,175.634,14.171,151.928
C02495=1098.527,-78.506,-49.053,175.635,14.172,151.928
C02496=1098.534,-78.257,-49.064,175.638,14.172,151.928
C02497=1098.539,-78.008,-49.074,175.639,14.172,151.927
C02498=1098.546,-77.757,-49.086,175.641,14.173,151.927
C02499=1098.551,-77.508,-49.097,175.643,14.173,151.927
C02500=1098.557,-77.258,-49.107,175.644,14.174,151.927
C02501=1098.563,-77.008,-49.118,175.646,14.174,151.926
C02502=1098.570,-76.758,-49.128,175.648,14.175,151.926
C02503=1098.575,-76.509,-49.139,175.650,14.175,151.926
C02504=1098.581,-76.259,-49.150,175.651,14.175,151.925
C02505=1098.587,-76.009,-49.161,175.653,14.176,151.925
C02506=1098.593,-75.760,-49.172,175.655,14.176,151.925
C02507=1098.599,-75.510,-49.183,175.657,14.177,151.924
C02508=1098.605,-75.260,-49.194,175.658,14.177,151.924
C02509=1098.612,-75.011,-49.205,175.660,14.178,151.924
C02510=1098.617,-74.761,-49.215,175.662,14.178,151.923
C02511=1098.623,-74.512,-49.226,175.664,14.179,151.923
C02512=1098.630,-74.262,-49.238,175.666,14.178,151.923
C02513=1098.635,-74.012,-49.248,175.668,14.179,151.922
C02514=1098.641,-73.763,-49.259,175.670,14.180,151.922
C02515=1098.647,-73.512,-49.271,175.671,14.181,151.922
C02516=1098.653,-73.263,-49.281,175.673,14.180,151.921
C02517=1098.659,-73.014,-49.292,175.675,14.181,151.921
C02518=1098.665,-72.764,-49.303,175.677,14.182,151.921
C02519=1098.671,-72.514,-49.314,175.679,14.182,151.920
C02520=1098.677,-72.264,-49.325,175.680,14.182,151.920
C02521=1098.682,-72.015,-49.336,175.682,14.183,151.920
C02522=1098.688,-71.765,-49.347,175.684,14.183,151.920
C02523=1098.694,-71.515,-49.358,175.686,14.184,151.919
C02524=1098.699,-71.265,-49.370,175.687,14.184,151.919
C02525=1098.705,-71.016,-49.381,175.689,14.185,151.919
C02526=1098.712,-70.766,-49.392,175.691,14.185,151.918
C02527=1098.717,-70.516,-49.403,175.693,14.186,151.918
C02528=1098.723,-70.267,-49.414,175.695,14.187,151.918
C02529=1098.729,-70.017,-49.425,175.696,14.186,151.917
C02530=1098.735,-69.767,-49.436,175.698,14.187,151.917
C02531=1098.741,-69.518,-49.447,175.700,14.188,151.917
C02532=1098.747,-69.268,-49.458,175.702,14.189,151.917
C02533=1098.753,-69.018,-49.469,175.703,14.188,151.916
C02534=1098.759,-68.769,-49.480,175.705,14.189,151.916
C02535=1098.765,-68.520,-49.491,175.707,14.190,151.916
C02536=1098.771,-68.269,-49.502,175.709,14.190,151.915
C02537=1098.776,-68.020,-49.514,175.711,14.191,151.915
C02538=1098.782,-67.770,-49.525,175.712,14.191,151.915
C02539=1098.788,-67.520,-49.536,175.714,14.191,151.914
C02540=1098.794,-67.270,-49.547,175.716,14.192,151.914
C02541=1098.800,-67.021,-49.558,175.718,14.193,151.914
C02542=1098.806,-66.771,-49.570,175.720,14.193,151.914
C02543=1098.812,-66.522,-49.581,175.721,14.193,151.913
C02544=1098.818,-66.272,-49.592,175.723,14.194,151.913
C02545=1098.824,-66.022,-49.603,175.725,14.195,151.913
C02546=1098.830,-65.773,-49.614,175.727,14.195,151.912
C02547=1098.836,-65.523,-49.626,175.729,14.196,151.912
C02548=1098.841,-65.273,-49.637,175.730,14.196,151.912
C02549=1098.847,-65.024,-49.648,175.733,14.196,151.911
C02550=1098.854,-64.755,-49.660,175.734,14.197,151.911
C02551=1098.860,-64.487,-49.672,175.736,14.198,151.911
C02552=1098.866,-64.218,-49.684,175.739,14.198,151.910
C02553=1098.873,-63.950,-49.697,175.740,14.199,151.910
C02554=1098.879,-63.700,-49.708,175.742,14.199,151.910
C02555=1098.885,-63.451,-49.719,175.745,14.200,151.909
C02556=1098.891,-63.200,-49.730,175.746,14.200,151.909
C02557=1098.897,-62.952,-49.741,175.747,14.201,151.909
C02558=1098.903,-62.701,-49.753,175.750,14.201,151.908
C02559=1098.908,-62.452,-49.764,175.752,14.202,151.908
C02560=1098.915,-62.201,-49.775,175.753,14.202,151.908
C02561=1098.921,-61.953,-49.787,175.755,14.202,151.908
C02562=1098.927,-61.703,-49.798,175.757,14.203,151.907
C02563=1098.933,-61.453,-49.809,175.759,14.204,151.907
C02564=1098.938,-61.204,-49.821,175.761,14.204,151.907
C02565=1098.945,-60.953,-49.833,175.763,14.205,151.906
C02566=1098.950,-60.704,-49.843,175.765,14.205,151.906
C02567=1098.957,-60.454,-49.855,175.766,14.206,151.906
C02568=1098.963,-60.205,-49.866,175.768,14.206,151.905
C02569=1098.968,-59.954,-49.878,175.770,14.207,151.905
C02570=1098.974,-59.706,-49.890,175.772,14.207,151.905
C02571=1098.980,-59.456,-49.901,175.774,14.208,151.904
C02572=1098.986,-59.206,-49.912,175.775,14.208,151.904
C02573=1098.992,-58.957,-49.923,175.777,14.209,151.904
C02574=1098.998,-58.707,-49.935,175.779,14.209,151.903
C02575=1099.004,-58.457,-49.946,175.781,14.210,151.903
C02576=1099.010,-58.207,-49.958,175.783,14.210,151.903
C02577=1099.016,-57.958,-49.969,175.785,14.211,151.903
C02578=1099.022,-57.708,-49.982,175.787,14.211,151.902
C02579=1099.028,-57.459,-49.992,175.788,14.211,151.902
C02580=1099.034,-57.208,-50.004,175.790,14.212,151.902
C02581=1099.040,-56.960,-50.015,175.792,14.213,151.901
C02582=1099.046,-56.709,-50.027,175.794,14.213,151.901
C02583=1099.052,-56.460,-50.039,175.796,14.214,151.901
C02584=1099.058,-56.210,-50.050,175.798,14.214,151.900
C02585=1099.064,-55.961,-50.062,175.799,14.214,151.900
C02586=1099.070,-55.711,-50.073,175.801,14.215,151.900
C02587=1099.076,-55.461,-50.085,175.803,14.216,151.899
C02588=1099.082,-55.212,-50.096,175.805,14.216,151.899
C02589=1099.089,-54.961,-50.107,175.807,14.217,151.899
C02590=1099.094,-54.712,-50.120,175.809,14.217,151.899
C02591=1099.100,-54.462,-50.131,175.811,14.218,151.898
C02592=1099.106,-54.213,-50.142,175.812,14.218,151.898
C02593=1099.113,-53.963,-50.154,175.814,14.219,151.898
C02594=1099.118,-53.714,-50.166,175.816,14.219,151.897
C02595=1099.124,-53.464,-50.177,175.818,14.220,151.897
C02596=1099.131,-53.214,-50.189,175.820,14.220,151.897
C02597=1099.136,-52.965,-50.201,175.822,14.221,151.896
C02598=1099.143,-52.715,-50.213,175.824,14.221,151.896
C02599=1099.149,-52.466,-50.224,175.825,14.222,151.896
C02600=1099.155,-52.216,-50.235,175.827,14.222,151.895
C02601=1099.160,-51.966,-50.248,175.829,14.223,151.895
C02602=1099.167,-51.716,-50.259,175.831,14.223,151.895
C02603=1099.173,-51.467,-50.271,175.833,14.224,151.894
C02604=1099.178,-51.217,-50.282,175.835,14.224,151.894
C02605=1099.185,-50.967,-50.294,175.837,14.225,151.894
C02606=1099.191,-50.718,-50.306,175.839,14.226,151.894
C02607=1099.197,-50.468,-50.318,175.841,14.226,151.893
C02608=1099.203,-50.218,-50.330,175.842,14.226,151.893
C02609=1099.208,-49.968,-50.341,175.844,14.227,151.893
C02610=1099.215,-49.719,-50.353,175.847,14.227,151.892
C02611=1099.220,-49.470,-50.365,175.848,14.228,151.892
C02612=1099.226,-49.220,-50.376,175.850,14.229,151.892
C02613=1099.232,-48.970,-50.389,175.852,14.230,151.891
C02614=1099.238,-48.703,-50.401,175.854,14.230,151.891
C02615=1099.245,-48.436,-50.414,175.856,14.231,151.891
C02616=1099.251,-48.169,-50.427,175.858,14.231,151.890
C02617=1099.257,-47.902,-50.439,175.860,14.232,151.890
C02618=1099.263,-47.652,-50.451,175.862,14.233,151.890
C02619=1099.269,-47.403,-50.463,175.864,14.233,151.889
C02620=1099.274,-47.152,-50.475,175.866,14.234,151.889
C02621=1099.281,-46.903,-50.487,175.868,14.234,151.889
C02622=1099.286,-46.654,-50.499,175.869,14.234,151.889
C02623=1099.292,-46.403,-50.510,175.871,14.235,151.888
C02624=1099.298,-46.154,-50.522,175.873,14.236,151.888
C02625=1099.304,-45.905,-50.534,175.875,14.236,151.888
C02626=1099.310,-45.654,-50.546,175.877,14.237,151.887
C02627=1099.316,-45.405,-50.558,175.879,14.237,151.887
C02628=1099.322,-45.155,-50.570,175.881,14.238,151.887
C02629=1099.327,-44.906,-50.583,175.883,14.239,151.886
C02630=1099.334,-44.656,-50.594,175.885,14.239,151.886
C02631=1099.340,-44.406,-50.606,175.887,14.240,151.886
C02632=1099.346,-44.157,-50.618,175.889,14.241,151.885
C02633=1099.351,-43.907,-50.631,175.890,14.241,151.885
C02634=1099.356,-43.658,-50.642,175.892,14.241,151.885
C02635=1099.363,-43.408,-50.654,175.894,14.242,151.885
C02636=1099.369,-43.158,-50.667,175.896,14.243,151.884
C02637=1099.375,-42.909,-50.678,175.898,14.243,151.884
C02638=1099.381,-42.659,-50.691,175.900,14.244,151.884
C02639=1099.387,-42.409,-50.703,175.902,14.244,151.883
C02640=1099.393,-42.160,-50.714,175.904,14.245,151.883
C02641=1099.399,-41.910,-50.727,175.906,14.246,151.883
C02642=1099.404,-41.660,-50.739,175.908,14.246,151.882
C02643=1099.410,-41.411,-50.751,175.910,14.247,151.882
C02644=1099.416,-41.161,-50.763,175.912,14.247,151.882
C02645=1099.423,-40.911,-50.775,175.914,14.248,151.881
C02646=1099.428,-40.662,-50.787,175.915,14.248,151.881
C02647=1099.434,-40.412,-50.799,175.917,14.249,151.881
C02648=1099.441,-40.163,-50.811,175.919,14.249,151.880
C02649=1099.446,-39.913,-50.824,175.921,14.250,151.880
C02650=1099.452,-39.664,-50.836,175.923,14.250,151.880
C02651=1099.458,-39.414,-50.848,175.925,14.251,151.880
C02652=1099.463,-39.164,-50.859,175.927,14.252,151.879
C02653=1099.469,-38.914,-50.872,175.929,14.252,151.879
C02654=1099.476,-38.665,-50.884,175.931,14.253,151.879
C02655=1099.481,-38.416,-50.896,175.933,14.254,151.878
C02656=1099.487,-38.166,-50.909,175.935,14.254,151.878
C02657=1099.493,-37.916,-50.921,175.937,14.255,151.878
C02658=1099.498,-37.667,-50.933,175.939,14.256,151.877
C02659=1099.505,-37.417,-50.945,175.941,14.256,151.877
C02660=1099.511,-37.167,-50.958,175.943,14.257,151.877
C02661=1099.516,-36.918,-50.970,175.945,14.257,151.876
C02662=1099.522,-36.668,-50.983,175.946,14.258,151.876
C02663=1099.528,-36.418,-50.995,175.949,14.258,151.876
C02664=1099.534,-36.169,-51.007,175.951,14.259,151.875
C02665=1099.540,-35.919,-51.019,175.952,14.260,151.875
C02666=1099.546,-35.670,-51.032,175.954,14.260,151.875
C02667=1099.552,-35.419,-51.044,175.956,14.260,151.875
C02668=1099.557,-35.170,-51.056,175.958,14.261,151.874
C02669=1099.563,-34.920,-51.069,175.960,14.261,151.874
C02670=1099.569,-34.670,-51.081,175.962,14.262,151.874
C02671=1099.575,-34.422,-51.093,175.964,14.263,151.873
C02672=1099.581,-34.172,-51.106,175.965,14.264,151.873
C02673=1099.587,-33.922,-51.119,175.968,14.264,151.873
C02674=1099.593,-33.672,-51.131,175.969,14.265,151.872
C02675=1099.598,-33.423,-51.143,175.971,14.266,151.872
C02676=1099.604,-33.173,-51.156,175.974,14.266,151.872
C02677=1099.611,-32.924,-51.168,175.975,14.267,151.871
C02678=1099.616,-32.657,-51.181,175.977,14.267,151.871
C02679=1099.623,-32.390,-51.194,175.979,14.268,151.871
C02680=1099.629,-32.123,-51.208,175.981,14.268,151.870
C02681=1099.636,-31.856,-51.221,175.984,14.269,151.870
C02682=1099.642,-31.607,-51.233,175.986,14.270,151.870
C02683=1099.647,-31.357,-51.246,175.988,14.271,151.869
C02684=1099.653,-31.107,-51.258,175.990,14.271,151.869
C02685=1099.659,-30.858,-51.271,175.992,14.272,151.869
C02686=1099.665,-30.608,-51.284,175.994,14.273,151.869
C02687=1099.671,-30.358,-51.296,175.996,14.273,151.868
C02688=1099.676,-30.109,-51.309,175.997,14.273,151.868
C02689=1099.682,-29.859,-51.321,175.999,14.274,151.868
C02690=1099.688,-29.609,-51.334,176.001,14.274,151.867
C02691=1099.695,-29.360,-51.346,176.003,14.275,151.867
C02692=1099.701,-29.110,-51.358,176.005,14.275,151.867
C02693=1099.706,-28.861,-51.371,176.007,14.276,151.866
C02694=1099.712,-28.612,-51.384,176.009,14.277,151.866
C02695=1099.718,-28.362,-51.396,176.011,14.277,151.866
C02696=1099.724,-28.112,-51.409,176.013,14.278,151.865
C02697=1099.730,-27.862,-51.421,176.015,14.279,151.865
C02698=1099.735,-27.613,-51.434,176.017,14.279,151.865
C02699=1099.741,-27.363,-51.447,176.019,14.280,151.864
C02700=1099.747,-27.114,-51.459,176.021,14.280,151.864
C02701=1099.753,-26.864,-51.472,176.023,14.281,151.864
C02702=1099.759,-26.614,-51.485,176.025,14.282,151.863
C02703=1099.765,-26.365,-51.497,176.027,14.282,151.863
C02704=1099.771,-26.115,-51.510,176.029,14.283,151.863
C02705=1099.776,-25.866,-51.523,176.031,14.283,151.862
C02706=1099.783,-25.616,-51.536,176.033,14.284,151.862
C02707=1099.789,-25.366,-51.548,176.035,14.285,151.862
C02708=1099.793,-25.117,-51.561,176.038,14.286,151.861
C02709=1099.799,-24.867,-51.574,176.040,14.287,151.861
C02710=1099.805,-24.618,-51.587,176.042,14.287,151.861
C02711=1099.811,-24.368,-51.600,176.044,14.288,151.861
C02712=1099.817,-24.118,-51.612,176.046,14.288,151.860
C02713=1099.823,-23.869,-51.625,176.048,14.289,151.860
C02714=1099.829,-23.620,-51.638,176.050,14.290,151.860
C02715=1099.834,-23.370,-51.650,176.052,14.290,151.859
C02716=1099.840,-23.120,-51.663,176.054,14.291,151.859
C02717=1099.846,-22.870,-51.677,176.056,14.291,151.859
C02718=1099.852,-22.620,-51.689,176.058,14.292,151.858
C02719=1099.858,-22.371,-51.702,176.060,14.292,151.858
C02720=1099.864,-22.121,-51.715,176.062,14.293,151.858
C02721=1099.869,-21.872,-51.727,176.064,14.294,151.857
C02722=1099.875,-21.623,-51.740,176.066,14.294,151.857
C02723=1099.881,-21.373,-51.753,176.067,14.295,151.857
C02724=1099.887,-21.123,-51.766,176.070,14.295,151.856
C02725=1099.893,-20.873,-51.779,176.072,14.296,151.856
C02726=1099.899,-20.623,-51.792,176.074,14.296,151.856
C02727=1099.905,-20.374,-51.805,176.076,14.297,151.855
C02728=1099.911,-20.124,-51.818,176.077,14.298,151.855
C02729=1099.916,-19.875,-51.830,176.080,14.298,151.855
C02730=1099.922,-19.626,-51.844,176.082,14.299,151.854
C02731=1099.927,-19.376,-51.856,176.084,14.299,151.854
C02732=1099.934,-19.126,-51.870,176.086,14.300,151.854
C02733=1099.940,-18.877,-51.882,176.087,14.301,151.853
C02734=1099.946,-18.627,-51.895,176.090,14.301,151.853
C02735=1099.951,-18.377,-51.909,176.092,14.302,151.853
C02736=1099.957,-18.128,-51.922,176.094,14.302,151.852
C02737=1099.963,-17.878,-51.934,176.096,14.303,151.852
C02738=1099.969,-17.629,-51.948,176.098,14.303,151.852
C02739=1099.975,-17.379,-51.960,176.100,14.304,151.851
C02740=1099.981,-17.129,-51.974,176.102,14.306,151.851
C02741=1099.987,-16.879,-51.987,176.105,14.306,151.851
C02742=1099.993,-16.612,-52.000,176.106,14.307,151.850
C02743=1099.999,-16.345,-52.014,176.109,14.307,151.850
C02744=1100.006,-16.077,-52.028,176.110,14.308,151.850
C02745=1100.012,-15.809,-52.042,176.113,14.308,151.849
C02746=1100.017,-15.560,-52.056,176.115,14.309,151.849
C02747=1100.024,-15.311,-52.069,176.117,14.309,151.849
C02748=1100.030,-15.061,-52.082,176.119,14.310,151.848
C02749=1100.035,-14.811,-52.095,176.122,14.311,151.848
C02750=1100.041,-14.561,-52.108,176.123,14.312,151.848
C02751=1100.047,-14.312,-52.121,176.126,14.312,151.847
C02752=1100.052,-14.062,-52.134,176.127,14.313,151.847
C02753=1100.058,-13.812,-52.148,176.129,14.313,151.847
C02754=1100.065,-13.563,-52.161,176.132,14.314,151.846
C02755=1100.069,-13.314,-52.174,176.133,14.314,151.846
C02756=1100.075,-13.064,-52.187,176.136,14.315,151.846
C02757=1100.081,-12.815,-52.201,176.137,14.316,151.845
C02758=1100.087,-12.565,-52.213,176.139,14.316,151.845
C02759=1100.093,-12.316,-52.227,176.142,14.317,151.845
C02760=1100.098,-12.066,-52.240,176.143,14.317,151.844
C02761=1100.104,-11.816,-52.253,176.146,14.318,151.844
C02762=1100.110,-11.567,-52.267,176.147,14.318,151.844
C02763=1100.116,-11.317,-52.280,176.150,14.319,151.843
C02764=1100.121,-11.067,-52.293,176.152,14.320,151.843
C02765=1100.128,-10.818,-52.307,176.155,14.320,151.843
C02766=1100.134,-10.569,-52.320,176.156,14.321,151.842
C02767=1100.139,-10.319,-52.333,176.158,14.322,151.842
C02768=1100.145,-10.069,-52.346,176.160,14.322,151.842
C02769=1100.151,-9.820,-52.360,176.162,14.323,151.841
C02770=1100.157,-9.570,-52.373,176.165,14.323,151.841
C02771=1100.162,-9.320,-52.387,176.166,14.324,151.841
C02772=1100.168,-9.071,-52.400,176.169,14.324,151.840
C02773=1100.174,-8.821,-52.414,176.170,14.325,151.840
C02774=1100.180,-8.571,-52.426,176.173,14.326,151.840
C02775=1100.186,-8.322,-52.440,176.175,14.327,151.839
C02776=1100.191,-8.073,-52.453,176.177,14.327,151.839
C02777=1100.198,-7.823,-52.467,176.179,14.328,151.839
C02778=1100.204,-7.573,-52.481,176.182,14.328,151.838
C02779=1100.209,-7.323,-52.494,176.183,14.329,151.838
C02780=1100.215,-7.074,-52.507,176.186,14.329,151.838
C02781=1100.221,-6.824,-52.521,176.187,14.330,151.837
C02782=1100.227,-6.575,-52.535,176.190,14.331,151.837
C02783=1100.233,-6.326,-52.548,176.192,14.331,151.837
C02784=1100.238,-6.075,-52.561,176.194,14.332,151.836
C02785=1100.244,-5.826,-52.574,176.196,14.332,151.836
C02786=1100.250,-5.577,-52.588,176.199,14.333,151.835
C02787=1100.256,-5.327,-52.601,176.200,14.334,151.835
C02788=1100.261,-5.078,-52.615,176.203,14.334,151.835
C02789=1100.268,-4.828,-52.629,176.204,14.335,151.834
C02790=1100.273,-4.579,-52.642,176.207,14.335,151.834
C02791=1100.280,-4.329,-52.656,176.209,14.336,151.834
C02792=1100.285,-4.079,-52.669,176.211,14.337,151.833
C02793=1100.291,-3.829,-52.682,176.213,14.337,151.833
C02794=1100.297,-3.580,-52.696,176.215,14.338,151.833
C02795=1100.303,-3.331,-52.710,176.217,14.338,151.832
C02796=1100.308,-3.081,-52.723,176.220,14.339,151.832
C02797=1100.314,-2.831,-52.737,176.222,14.340,151.832
C02798=1100.319,-2.582,-52.751,176.224,14.340,151.831
C02799=1100.326,-2.333,-52.764,176.226,14.341,151.831
C02800=1100.331,-2.083,-52.778,176.228,14.341,151.831
C02801=1100.337,-1.833,-52.792,176.230,14.342,151.830
C02802=1100.343,-1.584,-52.805,176.232,14.343,151.830
C02803=1100.349,-1.334,-52.820,176.234,14.343,151.830
C02804=1100.354,-1.084,-52.834,176.237,14.344,151.829
C02805=1100.360,-0.835,-52.847,176.239,14.345,151.829
C02806=1100.366,-0.566,-52.861,176.241,14.345,151.829
C02807=1100.372,-0.297,-52.876,176.243,14.346,151.828
C02808=1100.379,-0.027,-52.891,176.246,14.347,151.828
C02809=1100.384,0.242,-52.906,176.248,14.347,151.827
C02810=1100.391,0.492,-52.920,176.250,14.348,151.827
C02811=1100.396,0.741,-52.934,176.252,14.348,151.827
C02812=1100.402,0.991,-52.947,176.254,14.349,151.826
C02813=1100.407,1.240,-52.961,176.256,14.350,151.826
C02814=1100.413,1.490,-52.975,176.258,14.350,151.826
C02815=1100.419,1.739,-52.988,176.261,14.351,151.825
C02816=1100.425,1.989,-53.003,176.263,14.352,151.825
C02817=1100.430,2.239,-53.017,176.265,14.352,151.824
C02818=1100.436,2.489,-53.030,176.267,14.353,151.824
C02819=1100.442,2.737,-53.044,176.269,14.353,151.824
C02820=1100.448,2.987,-53.058,176.271,14.354,151.824
C02821=1100.453,3.236,-53.072,176.273,14.354,151.823
C02822=1100.459,3.487,-53.086,176.276,14.355,151.823
C02823=1100.465,3.736,-53.100,176.278,14.356,151.822
C02824=1100.471,3.985,-53.113,176.280,14.356,151.822
C02825=1100.477,4.235,-53.127,176.282,14.357,151.822
C02826=1100.482,4.485,-53.141,176.284,14.357,151.821
C02827=1100.488,4.734,-53.156,176.287,14.358,151.821
C02828=1100.494,4.984,-53.170,176.288,14.358,151.821
C02829=1100.500,5.233,-53.183,176.291,14.359,151.820
C02830=1100.506,5.483,-53.197,176.294,14.360,151.820
C02831=1100.511,5.732,-53.211,176.295,14.360,151.819
C02832=1100.517,5.981,-53.226,176.298,14.361,151.819
C02833=1100.523,6.231,-53.240,176.299,14.361,151.819
C02834=1100.528,6.481,-53.254,176.302,14.362,151.818
C02835=1100.535,6.730,-53.267,176.304,14.362,151.818
C02836=1100.540,6.980,-53.281,176.306,14.363,151.818
C02837=1100.546,7.230,-53.296,176.309,14.364,151.817
C02838=1100.552,7.479,-53.310,176.311,14.364,151.817
C02839=1100.557,7.729,-53.323,176.313,14.365,151.817
C02840=1100.563,7.978,-53.337,176.315,14.365,151.816
C02841=1100.569,8.227,-53.352,176.317,14.365,151.816
C02842=1100.575,8.477,-53.366,176.319,14.366,151.815
C02843=1100.581,8.727,-53.379,176.322,14.367,151.815
C02844=1100.587,8.976,-53.394,176.324,14.367,151.815
C02845=1100.593,9.226,-53.408,176.326,14.368,151.814
C02846=1100.598,9.476,-53.422,176.328,14.369,151.814
C02847=1100.604,9.725,-53.437,176.330,14.369,151.813
C02848=1100.610,9.974,-53.451,176.333,14.369,151.813
C02849=1100.616,10.224,-53.465,176.334,14.370,151.813
C02850=1100.621,10.473,-53.479,176.337,14.371,151.812
C02851=1100.628,10.723,-53.493,176.340,14.371,151.812
C02852=1100.634,10.973,-53.507,176.342,14.372,151.811
C02853=1100.639,11.222,-53.521,176.344,14.372,151.811
C02854=1100.645,11.471,-53.535,176.346,14.373,151.811
C02855=1100.650,11.721,-53.549,176.348,14.373,151.810
C02856=1100.657,11.971,-53.564,176.351,14.374,151.810
C02857=1100.662,12.220,-53.578,176.353,14.375,151.810
C02858=1100.668,12.469,-53.593,176.355,14.375,151.809
C02859=1100.674,12.719,-53.607,176.357,14.375,151.809
C02860=1100.680,12.969,-53.621,176.359,14.376,151.808
C02861=1100.685,13.218,-53.635,176.361,14.376,151.808
C02862=1100.691,13.468,-53.649,176.364,14.377,151.808
C02863=1100.697,13.717,-53.664,176.366,14.378,151.807
C02864=1100.703,13.968,-53.678,176.369,14.378,151.807
C02865=1100.709,14.216,-53.693,176.371,14.378,151.806
C02866=1100.715,14.466,-53.707,176.373,14.379,151.806
C02867=1100.720,14.715,-53.721,176.375,14.379,151.806
C02868=1100.726,14.965,-53.736,176.378,14.380,151.805
C02869=1100.732,15.214,-53.750,176.380,14.381,151.805
C02870=1100.739,15.486,-53.766,176.382,14.381,151.805
C02871=1100.744,15.757,-53.781,176.385,14.382,151.804
C02872=1100.751,16.029,-53.797,176.387,14.383,151.804
C02873=1100.757,16.299,-53.812,176.389,14.383,151.803
C02874=1100.764,16.549,-53.827,176.392,14.383,151.803
C02875=1100.769,16.799,-53.841,176.394,14.384,151.802
C02876=1100.774,17.048,-53.856,176.397,14.385,151.802
C02877=1100.780,17.298,-53.871,176.399,14.385,151.802
C02878=1100.786,17.547,-53.885,176.401,14.386,151.801
C02879=1100.792,17.796,-53.899,176.403,14.386,151.801
C02880=1100.798,18.046,-53.914,176.406,14.387,151.800
C02881=1100.804,18.295,-53.928,176.408,14.387,151.800
C02882=1100.809,18.545,-53.942,176.410,14.388,151.800
C02883=1100.815,18.795,-53.958,176.412,14.388,151.799
C02884=1100.820,19.044,-53.972,176.414,14.389,151.799
C02885=1100.827,19.294,-53.986,176.417,14.390,151.799
C02886=1100.832,19.543,-54.001,176.419,14.390,151.798
C02887=1100.838,19.792,-54.016,176.422,14.390,151.798
C02888=1100.844,20.042,-54.030,176.424,14.391,151.797
C02889=1100.849,20.292,-54.045,176.426,14.391,151.797
C02890=1100.856,20.541,-54.060,176.429,14.392,151.797
C02891=1100.861,20.791,-54.074,176.431,14.393,151.796
C02892=1100.867,21.040,-54.088,176.433,14.393,151.796
C02893=1100.873,21.290,-54.104,176.435,14.393,151.795
C02894=1100.878,21.539,-54.118,176.437,14.394,151.795
C02895=1100.884,21.788,-54.132,176.440,14.395,151.795
C02896=1100.890,22.038,-54.147,176.442,14.395,151.794
C02897=1100.895,22.288,-54.162,176.444,14.396,151.794
C02898=1100.901,22.537,-54.177,176.447,14.396,151.793
C02899=1100.907,22.786,-54.191,176.449,14.396,151.793
C02900=1100.913,23.036,-54.206,176.452,14.397,151.792
C02901=1100.918,23.286,-54.221,176.454,14.398,151.792
C02902=1100.924,23.535,-54.235,176.456,14.398,151.792
C02903=1100.930,23.785,-54.250,176.458,14.399,151.791
C02904=1100.935,24.034,-54.265,176.460,14.399,151.791
C02905=1100.941,24.284,-54.280,176.463,14.400,151.790
C02906=1100.947,24.533,-54.294,176.465,14.400,151.790
C02907=1100.953,24.783,-54.310,176.468,14.401,151.790
C02908=1100.959,25.032,-54.324,176.470,14.401,151.789
C02909=1100.965,25.282,-54.339,176.472,14.401,151.789
C02910=1100.970,25.532,-54.354,176.475,14.402,151.788
C02911=1100.976,25.781,-54.369,176.477,14.402,151.788
C02912=1100.982,26.030,-54.383,176.479,14.403,151.787
C02913=1100.988,26.280,-54.398,176.482,14.403,151.787
C02914=1100.993,26.529,-54.413,176.484,14.404,151.787
C02915=1100.999,26.778,-54.428,176.487,14.404,151.786
C02916=1101.005,27.028,-54.443,176.489,14.405,151.786
C02917=1101.010,27.278,-54.457,176.491,14.405,151.785
C02918=1101.017,27.527,-54.472,176.493,14.406,151.785
C02919=1101.022,27.776,-54.487,176.496,14.407,151.785
C02920=1101.028,28.026,-54.502,176.498,14.407,151.784
C02921=1101.034,28.275,-54.517,176.500,14.407,151.784
C02922=1101.040,28.525,-54.533,176.502,14.408,151.783
C02923=1101.046,28.775,-54.547,176.505,14.409,151.783
C02924=1101.051,29.024,-54.563,176.508,14.409,151.783
C02925=1101.057,29.273,-54.577,176.510,14.409,151.782
C02926=1101.062,29.523,-54.593,176.512,14.410,151.782
C02927=1101.068,29.772,-54.607,176.514,14.410,151.781
C02928=1101.074,30.022,-54.623,176.517,14.411,151.781
C02929=1101.080,30.271,-54.637,176.519,14.411,151.780
C02930=1101.085,30.521,-54.653,176.522,14.412,151.780
C02931=1101.091,30.770,-54.668,176.524,14.412,151.780
C02932=1101.097,31.020,-54.683,176.527,14.413,151.779
C02933=1101.103,31.269,-54.698,176.529,14.413,151.779
C02934=1101.109,31.542,-54.714,176.531,14.413,151.778
C02935=1101.115,31.814,-54.731,176.534,14.414,151.778
C02936=1101.121,32.087,-54.747,176.537,14.414,151.777
C02937=1101.128,32.360,-54.763,176.539,14.415,151.777
C02938=1101.133,32.609,-54.779,176.542,14.416,151.776
C02939=1101.139,32.859,-54.794,176.544,14.416,151.776
C02940=1101.145,33.109,-54.809,176.546,14.416,151.776
C02941=1101.151,33.358,-54.824,176.549,14.417,151.775
C02942=1101.157,33.607,-54.840,176.552,14.417,151.774
C02943=1101.162,33.856,-54.855,176.554,14.417,151.774
C02944=1101.168,34.106,-54.870,176.556,14.418,151.774
C02945=1101.173,34.355,-54.885,176.559,14.419,151.773
C02946=1101.179,34.605,-54.900,176.561,14.419,151.773
C02947=1101.185,34.855,-54.916,176.563,14.419,151.772
C02948=1101.191,35.104,-54.930,176.565,14.420,151.772
C02949=1101.196,35.354,-54.946,176.568,14.421,151.771
C02950=1101.202,35.603,-54.962,176.571,14.421,151.771
C02951=1101.208,35.852,-54.977,176.573,14.421,151.770
C02952=1101.214,36.102,-54.992,176.575,14.421,151.770
C02953=1101.220,36.351,-55.007,176.578,14.422,151.770
C02954=1101.225,36.601,-55.022,176.580,14.422,151.769
C02955=1101.231,36.851,-55.038,176.583,14.423,151.769
C02956=1101.237,37.099,-55.053,176.585,14.423,151.768
C02957=1101.243,37.349,-55.069,176.588,14.424,151.768
C02958=1101.248,37.598,-55.083,176.590,14.424,151.767
C02959=1101.254,37.848,-55.099,176.592,14.424,151.767
C02960=1101.260,38.098,-55.115,176.595,14.425,151.766
C02961=1101.266,38.347,-55.130,176.598,14.425,151.766
C02962=1101.271,38.597,-55.145,176.600,14.426,151.766
C02963=1101.277,38.847,-55.161,176.602,14.426,151.765
C02964=1101.282,39.095,-55.177,176.605,14.426,151.765
C02965=1101.289,39.345,-55.192,176.607,14.427,151.764
C02966=1101.294,39.594,-55.207,176.610,14.427,151.764
C02967=1101.300,39.844,-55.222,176.612,14.428,151.763
C02968=1101.305,40.093,-55.239,176.615,14.429,151.763
C02969=1101.311,40.342,-55.253,176.617,14.428,151.762
C02970=1101.317,40.592,-55.269,176.620,14.429,151.762
C02971=1101.323,40.842,-55.285,176.622,14.429,151.761
C02972=1101.328,41.091,-55.300,176.625,14.430,151.761
C02973=1101.334,41.341,-55.316,176.627,14.430,151.761
C02974=1101.340,41.590,-55.331,176.629,14.430,151.760
C02975=1101.345,41.839,-55.346,176.632,14.431,151.760
C02976=1101.351,42.089,-55.362,176.635,14.432,151.759
C02977=1101.357,42.339,-55.378,176.637,14.432,151.759
C02978=1101.362,42.588,-55.393,176.639,14.432,151.758
C02979=1101.369,42.837,-55.409,176.642,14.433,151.758
C02980=1101.374,43.087,-55.425,176.644,14.433,151.757
C02981=1101.379,43.336,-55.440,176.647,14.433,151.757
C02982=1101.385,43.585,-55.456,176.649,14.433,151.756
C02983=1101.391,43.835,-55.472,176.652,14.434,151.756
C02984=1101.397,44.085,-55.488,176.654,14.435,151.755
C02985=1101.403,44.334,-55.502,176.656,14.435,151.755
C02986=1101.409,44.583,-55.519,176.660,14.435,151.754
C02987=1101.414,44.833,-55.534,176.662,14.436,151.754
C02988=1101.419,45.082,-55.549,176.664,14.436,151.754
C02989=1101.425,45.332,-55.566,176.666,14.436,151.753
C02990=1101.431,45.582,-55.581,176.670,14.437,151.752
C02991=1101.436,45.830,-55.597,176.672,14.437,151.752
C02992=1101.442,46.080,-55.613,176.674,14.438,151.752
C02993=1101.448,46.330,-55.629,176.677,14.438,151.751
C02994=1101.453,46.579,-55.644,176.679,14.438,151.751
C02995=1101.459,46.828,-55.660,176.682,14.439,151.750
C02996=1101.464,47.078,-55.676,176.684,14.439,151.750
C02997=1101.470,47.327,-55.692,176.687,14.440,151.749
C02998=1101.476,47.600,-55.709,176.689,14.440,151.749
C02999=1101.482,47.873,-55.727,176.693,14.440,151.748
C03000=1101.488,48.145,-55.745,176.695,14.441,151.748
C03001=1101.495,48.418,-55.761,176.698,14.441,151.747
C03002=1101.501,48.668,-55.777,176.700,14.442,151.747
C03003=1101.505,48.917,-55.793,176.703,14.441,151.746
C03004=1101.511,49.166,-55.809,176.706,14.442,151.746
C03005=1101.517,49.416,-55.825,176.708,14.443,151.745
C03006=1101.523,49.665,-55.841,176.710,14.443,151.745
C03007=1101.528,49.914,-55.856,176.713,14.444,151.744
C03008=1101.534,50.164,-55.873,176.716,14.444,151.744
C03009=1101.540,50.413,-55.889,176.718,14.444,151.743
C03010=1101.545,50.663,-55.905,176.720,14.444,151.743
C03011=1101.551,50.912,-55.921,176.723,14.445,151.742
C03012=1101.557,51.161,-55.937,176.726,14.445,151.742
C03013=1101.562,51.411,-55.952,176.728,14.445,151.741
C03014=1101.568,51.660,-55.968,176.731,14.446,151.741
C03015=1101.574,51.910,-55.985,176.733,14.446,151.740
C03016=1101.580,52.159,-56.001,176.736,14.446,151.740
C03017=1101.585,52.408,-56.016,176.739,14.447,151.739
C03018=1101.591,52.658,-56.032,176.741,14.447,151.739
C03019=1101.597,52.907,-56.049,176.744,14.447,151.738
C03020=1101.602,53.157,-56.066,176.746,14.447,151.738
C03021=1101.608,53.407,-56.081,176.749,14.448,151.737
C03022=1101.614,53.656,-56.097,176.751,14.448,151.737
C03023=1101.619,53.905,-56.113,176.754,14.448,151.736
C03024=1101.625,54.154,-56.129,176.757,14.449,151.736
C03025=1101.631,54.404,-56.145,176.759,14.449,151.735
C03026=1101.637,54.653,-56.161,176.762,14.449,151.735
C03027=1101.643,54.903,-56.177,176.765,14.450,151.734
C03028=1101.649,55.152,-56.194,176.767,14.450,151.734
C03029=1101.654,55.402,-56.211,176.769,14.450,151.733
C03030=1101.660,55.651,-56.227,176.773,14.451,151.733
C03031=1101.665,55.900,-56.242,176.775,14.451,151.732
C03032=1101.671,56.150,-56.258,176.777,14.451,151.732
C03033=1101.677,56.399,-56.275,176.781,14.451,151.731
C03034=1101.683,56.648,-56.291,176.783,14.452,151.731
C03035=1101.689,56.898,-56.307,176.785,14.452,151.730
C03036=1101.694,57.147,-56.324,176.787,14.452,151.730
C03037=1101.700,57.397,-56.340,176.791,14.452,151.729
C03038=1101.706,57.646,-56.356,176.793,14.452,151.728
C03039=1101.712,57.896,-56.372,176.795,14.453,151.728
C03040=1101.718,58.145,-56.388,176.799,14.453,151.727
C03041=1101.723,58.395,-56.405,176.801,14.453,151.727
C03042=1101.729,58.644,-56.421,176.803,14.453,151.726
C03043=1101.735,58.894,-56.438,176.807,14.454,151.726
C03044=1101.740,59.142,-56.453,176.809,14.454,151.725
C03045=1101.746,59.392,-56.470,176.811,14.454,151.725
C03046=1101.751,59.641,-56.487,176.815,14.455,151.724
C03047=1101.757,59.891,-56.503,176.817,14.455,151.724
C03048=1101.763,60.140,-56.519,176.819,14.455,151.723
C03049=1101.769,60.389,-56.535,176.823,14.455,151.722
C03050=1101.775,60.639,-56.552,176.825,14.455,151.722
C03051=1101.780,60.888,-56.568,176.827,14.456,151.721
C03052=1101.786,61.138,-56.585,176.831,14.456,151.721
C03053=1101.792,61.387,-56.601,176.833,14.456,151.720
C03054=1101.798,61.637,-56.617,176.836,14.456,151.720
C03055=1101.803,61.886,-56.634,176.839,14.457,151.719
C03056=1101.810,62.135,-56.651,176.841,14.457,151.719
C03057=1101.815,62.384,-56.667,176.844,14.457,151.718
C03058=1101.821,62.634,-56.684,176.846,14.456,151.718
C03059=1101.827,62.883,-56.700,176.849,14.457,151.717
C03060=1101.833,63.133,-56.717,176.852,14.457,151.717
C03061=1101.839,63.383,-56.733,176.854,14.457,151.716
C03062=1101.845,63.655,-56.751,176.857,14.458,151.715
C03063=1101.852,63.927,-56.769,176.861,14.458,151.715
C03064=1101.858,64.199,-56.787,176.863,14.458,151.714
C03065=1101.865,64.472,-56.805,176.867,14.459,151.713
C03066=1101.870,64.722,-56.822,176.869,14.459,151.713
C03067=1101.876,64.971,-56.839,176.872,14.458,151.712
C03068=1101.881,65.221,-56.855,176.875,14.459,151.712
C03069=1101.887,65.469,-56.872,176.877,14.459,151.711
C03070=1101.892,65.719,-56.889,176.880,14.459,151.711
C03071=1101.898,65.968,-56.906,176.883,14.460,151.710
C03072=1101.904,66.218,-56.922,176.885,14.460,151.710
C03073=1101.910,66.467,-56.939,176.888,14.459,151.709
C03074=1101.916,66.716,-56.956,176.891,14.460,151.709
C03075=1101.921,66.966,-56.972,176.893,14.460,151.708
C03076=1101.927,67.215,-56.989,176.896,14.460,151.707
C03077=1101.932,67.465,-57.006,176.899,14.461,151.707
C03078=1101.939,67.713,-57.023,176.902,14.461,151.706
C03079=1101.944,67.963,-57.039,176.904,14.461,151.706
C03080=1101.950,68.212,-57.056,176.907,14.461,151.705
C03081=1101.955,68.462,-57.072,176.910,14.461,151.705
C03082=1101.961,68.711,-57.089,176.912,14.461,151.704
C03083=1101.967,68.961,-57.107,176.915,14.462,151.703
C03084=1101.973,69.211,-57.123,176.918,14.462,151.703
C03085=1101.978,69.460,-57.140,176.920,14.462,151.702
C03086=1101.984,69.709,-57.157,176.924,14.462,151.702
C03087=1101.990,69.959,-57.174,176.926,14.462,151.701
C03088=1101.996,70.207,-57.191,176.929,14.462,151.700
C03089=1102.001,70.457,-57.207,176.932,14.462,151.700
C03090=1102.007,70.706,-57.225,176.934,14.463,151.699
C03091=1102.013,70.955,-57.241,176.937,14.463,151.699
C03092=1102.018,71.205,-57.258,176.940,14.463,151.698
C03093=1102.024,71.454,-57.275,176.942,14.463,151.698
C03094=1102.029,71.703,-57.292,176.946,14.464,151.697
C03095=1102.035,71.953,-57.310,176.948,14.464,151.696
C03096=1102.041,72.203,-57.326,176.951,14.463,151.696
C03097=1102.046,72.452,-57.343,176.954,14.464,151.695
C03098=1102.052,72.701,-57.361,176.957,14.464,151.695
C03099=1102.058,72.951,-57.377,176.959,14.464,151.694
C03100=1102.063,73.200,-57.394,176.962,14.464,151.693
C03101=1102.069,73.449,-57.411,176.965,14.464,151.693
C03102=1102.075,73.698,-57.428,176.967,14.464,151.692
C03103=1102.081,73.948,-57.445,176.971,14.465,151.692
C03104=1102.086,74.197,-57.463,176.973,14.464,151.691
C03105=1102.092,74.447,-57.479,176.976,14.464,151.691
C03106=1102.098,74.696,-57.497,176.979,14.465,151.690
C03107=1102.103,74.945,-57.514,176.981,14.465,151.689
C03108=1102.109,75.194,-57.531,176.985,14.465,151.689
C03109=1102.115,75.445,-57.548,176.987,14.465,151.688
C03110=1102.121,75.694,-57.565,176.990,14.465,151.688
C03111=1102.126,75.943,-57.582,176.993,14.466,151.687
C03112=1102.132,76.192,-57.599,176.996,14.466,151.686
C03113=1102.138,76.441,-57.617,176.998,14.465,151.686
C03114=1102.143,76.691,-57.634,177.002,14.465,151.685
C03115=1102.150,76.940,-57.651,177.004,14.465,151.684
C03116=1102.155,77.190,-57.668,177.007,14.465,151.684
C03117=1102.160,77.439,-57.685,177.010,14.466,151.683
C03118=1102.167,77.687,-57.702,177.012,14.466,151.683
C03119=1102.172,77.938,-57.720,177.016,14.466,151.682
C03120=1102.178,78.187,-57.737,177.018,14.466,151.682
C03121=1102.183,78.436,-57.755,177.021,14.466,151.681
C03122=1102.189,78.686,-57.772,177.024,14.466,151.680
C03123=1102.195,78.934,-57.789,177.027,14.466,151.680
C03124=1102.201,79.184,-57.806,177.029,14.466,151.679
C03125=1102.206,79.434,-57.823,177.033,14.466,151.678
C03126=1102.212,79.706,-57.843,177.035,14.466,151.678
C03127=1102.218,79.979,-57.861,177.039,14.466,151.677
C03128=1102.225,80.250,-57.880,177.042,14.467,151.676
C03129=1102.231,80.523,-57.900,177.045,14.466,151.676
C03130=1102.236,80.772,-57.917,177.048,14.467,151.675
C03131=1102.242,81.021,-57.934,177.051,14.467,151.675
C03132=1102.247,81.270,-57.952,177.053,14.467,151.674
C03133=1102.253,81.520,-57.970,177.056,14.467,151.673
C03134=1102.259,81.770,-57.987,177.059,14.467,151.673
C03135=1102.264,82.019,-58.004,177.062,14.467,151.672
C03136=1102.270,82.268,-58.021,177.065,14.467,151.671
C03137=1102.277,82.517,-58.039,177.068,14.467,151.671
C03138=1102.282,82.766,-58.057,177.071,14.468,151.670
C03139=1102.287,83.016,-58.073,177.074,14.467,151.669
C03140=1102.293,83.265,-58.091,177.076,14.467,151.669
C03141=1102.299,83.515,-58.109,177.080,14.467,151.668
C03142=1102.304,83.764,-58.127,177.082,14.467,151.668
C03143=1102.310,84.013,-58.144,177.085,14.467,151.667
C03144=1102.316,84.263,-58.162,177.088,14.467,151.666
C03145=1102.322,84.512,-58.180,177.091,14.467,151.666
C03146=1102.327,84.761,-58.196,177.094,14.467,151.665
C03147=1102.332,85.010,-58.214,177.097,14.467,151.664
C03148=1102.338,85.260,-58.232,177.099,14.467,151.664
C03149=1102.344,85.509,-58.249,177.103,14.467,151.663
C03150=1102.349,85.758,-58.267,177.105,14.467,151.662
C03151=1102.356,86.008,-58.285,177.108,14.467,151.662
C03152=1102.361,86.257,-58.303,177.111,14.467,151.661
C03153=1102.367,86.506,-58.320,177.114,14.467,151.661
C03154=1102.373,86.756,-58.338,177.117,14.468,151.660
C03155=1102.378,87.005,-58.356,177.120,14.467,151.659
C03156=1102.384,87.255,-58.374,177.123,14.467,151.659
C03157=1102.390,87.504,-58.391,177.126,14.467,151.658
C03158=1102.395,87.753,-58.409,177.129,14.467,151.657
C03159=1102.402,88.002,-58.427,177.132,14.468,151.657
C03160=1102.407,88.251,-58.444,177.135,14.467,151.656
C03161=1102.413,88.501,-58.462,177.137,14.467,151.655
C03162=1102.419,88.750,-58.480,177.141,14.467,151.655
C03163=1102.424,88.999,-58.497,177.143,14.467,151.654
C03164=1102.430,89.249,-58.515,177.146,14.466,151.653
C03165=1102.436,89.498,-58.533,177.150,14.467,151.653
C03166=1102.441,89.747,-58.551,177.152,14.466,151.652
C03167=1102.447,89.997,-58.569,177.156,14.467,151.651
C03168=1102.452,90.246,-58.586,177.159,14.466,151.651
C03169=1102.459,90.495,-58.605,177.161,14.466,151.650
C03170=1102.464,90.744,-58.623,177.165,14.466,151.649
C03171=1102.470,90.994,-58.641,177.167,14.466,151.649
C03172=1102.476,91.243,-58.658,177.171,14.466,151.648
C03173=1102.481,91.492,-58.676,177.173,14.466,151.647
C03174=1102.487,91.742,-58.694,177.176,14.466,151.647
C03175=1102.492,91.991,-58.712,177.179,14.466,151.646
C03176=1102.498,92.240,-58.730,177.182,14.466,151.645
C03177=1102.504,92.489,-58.748,177.185,14.466,151.645
C03178=1102.509,92.739,-58.766,177.188,14.466,151.644
C03179=1102.515,92.989,-58.784,177.191,14.466,151.643
C03180=1102.521,93.238,-58.802,177.194,14.466,151.643
C03181=1102.527,93.487,-58.820,177.197,14.466,151.642
C03182=1102.532,93.736,-58.838,177.201,14.466,151.641
C03183=1102.537,93.985,-58.856,177.203,14.466,151.641
C03184=1102.543,94.235,-58.874,177.206,14.465,151.640
C03185=1102.549,94.484,-58.892,177.209,14.466,151.639
C03186=1102.555,94.733,-58.911,177.212,14.465,151.638
C03187=1102.560,94.982,-58.928,177.216,14.465,151.638
C03188=1102.566,95.232,-58.946,177.218,14.465,151.637
C03189=1102.571,95.481,-58.965,177.221,14.465,151.636
C03190=1102.578,95.753,-58.985,177.225,14.465,151.636
C03191=1102.584,96.026,-59.004,177.228,14.465,151.635
C03192=1102.591,96.298,-59.024,177.231,14.464,151.634
C03193=1102.597,96.571,-59.044,177.235,14.464,151.633
C03194=1102.602,96.820,-59.063,177.237,14.464,151.633
C03195=1102.608,97.069,-59.080,177.241,14.464,151.632
C03196=1102.614,97.318,-59.098,177.244,14.464,151.631
C03197=1102.619,97.568,-59.117,177.246,14.464,151.631
C03198=1102.625,97.817,-59.135,177.250,14.464,151.630
C03199=1102.631,98.066,-59.154,177.252,14.463,151.629
C03200=1102.636,98.315,-59.172,177.256,14.463,151.628
C03201=1102.642,98.565,-59.190,177.259,14.463,151.628
C03202=1102.648,98.814,-59.208,177.261,14.463,151.627
C03203=1102.653,99.064,-59.226,177.265,14.463,151.626
C03204=1102.659,99.312,-59.245,177.268,14.462,151.626
C03205=1102.665,99.562,-59.263,177.271,14.463,151.625
C03206=1102.670,99.810,-59.282,177.274,14.462,151.624
C03207=1102.677,100.060,-59.299,177.277,14.462,151.623
C03208=1102.682,100.310,-59.319,177.280,14.462,151.623
C03209=1102.688,100.559,-59.336,177.283,14.462,151.622
C03210=1102.694,100.808,-59.355,177.286,14.462,151.621
C03211=1102.699,101.057,-59.373,177.289,14.462,151.621
C03212=1102.705,101.306,-59.392,177.292,14.461,151.620
C03213=1102.710,101.556,-59.410,177.296,14.461,151.619
C03214=1102.717,101.805,-59.429,177.298,14.461,151.619
C03215=1102.722,102.055,-59.447,177.302,14.461,151.618
C03216=1102.728,102.303,-59.465,177.305,14.461,151.617
C03217=1102.733,102.553,-59.484,177.308,14.461,151.616
C03218=1102.738,102.802,-59.503,177.311,14.460,151.616
C03219=1102.745,103.051,-59.521,177.314,14.460,151.615
C03220=1102.750,103.301,-59.540,177.317,14.460,151.614
C03221=1102.756,103.550,-59.558,177.320,14.460,151.613
C03222=1102.761,103.800,-59.577,177.324,14.460,151.613
C03223=1102.767,104.048,-59.595,177.327,14.459,151.612
C03224=1102.773,104.298,-59.614,177.329,14.459,151.611
C03225=1102.778,104.547,-59.632,177.333,14.459,151.610
C03226=1102.784,104.796,-59.651,177.335,14.459,151.610
C03227=1102.790,105.045,-59.670,177.339,14.459,151.609
C03228=1102.795,105.294,-59.688,177.342,14.458,151.608
C03229=1102.801,105.544,-59.707,177.345,14.459,151.608
C03230=1102.807,105.792,-59.725,177.348,14.458,151.607
C03231=1102.812,106.042,-59.744,177.351,14.458,151.606
C03232=1102.818,106.292,-59.763,177.355,14.458,151.605
C03233=1102.824,106.540,-59.781,177.358,14.457,151.605
C03234=1102.829,106.790,-59.801,177.361,14.457,151.604
C03235=1102.835,107.039,-59.819,177.364,14.457,151.603
C03236=1102.841,107.288,-59.837,177.367,14.456,151.602
C03237=1102.846,107.538,-59.857,177.370,14.456,151.602
C03238=1102.853,107.787,-59.875,177.373,14.456,151.601
C03239=1102.857,108.036,-59.894,177.377,14.456,151.600
C03240=1102.863,108.285,-59.913,177.380,14.455,151.599
C03241=1102.870,108.535,-59.931,177.383,14.455,151.599
C03242=1102.875,108.783,-59.950,177.386,14.455,151.598
C03243=1102.880,109.033,-59.970,177.389,14.454,151.597
C03244=1102.886,109.283,-59.987,177.393,14.455,151.596
C03245=1102.892,109.532,-60.007,177.395,14.454,151.596
C03246=1102.897,109.781,-60.026,177.399,14.454,151.595
C03247=1102.904,110.030,-60.044,177.402,14.454,151.594
C03248=1102.909,110.279,-60.064,177.405,14.453,151.593
C03249=1102.914,110.528,-60.082,177.409,14.453,151.592
C03250=1102.921,110.777,-60.101,177.411,14.452,151.592
C03251=1102.927,111.027,-60.120,177.415,14.452,151.591
C03252=1102.932,111.277,-60.139,177.418,14.452,151.590
C03253=1102.937,111.525,-60.158,177.421,14.452,151.589
C03254=1102.944,111.798,-60.178,177.425,14.451,151.588
C03255=1102.950,112.070,-60.199,177.428,14.451,151.588
C03256=1102.956,112.342,-60.220,177.432,14.451,151.587
C03257=1102.962,112.615,-60.241,177.435,14.450,151.586
C03258=1102.969,112.864,-60.260,177.439,14.451,151.585
C03259=1102.974,113.113,-60.279,177.441,14.450,151.584
C03260=1102.980,113.363,-60.298,177.445,14.449,151.584
C03261=1102.985,113.611,-60.317,177.448,14.449,151.583
C03262=1102.991,113.861,-60.336,177.451,14.449,151.582
C03263=1102.997,114.110,-60.355,177.455,14.449,151.581
C03264=1103.003,114.359,-60.374,177.457,14.448,151.581
C03265=1103.008,114.608,-60.393,177.461,14.448,151.580
C03266=1103.014,114.857,-60.412,177.464,14.447,151.579
C03267=1103.019,115.107,-60.432,177.467,14.447,151.578
C03268=1103.025,115.356,-60.451,177.471,14.447,151.577
C03269=1103.030,115.605,-60.470,177.473,14.447,151.577
C03270=1103.036,115.854,-60.489,177.477,14.447,151.576
C03271=1103.041,116.104,-60.508,177.480,14.446,151.575
C03272=1103.047,116.353,-60.528,177.484,14.446,151.574
C03273=1103.052,116.602,-60.546,177.487,14.445,151.573
C03274=1103.058,116.852,-60.566,177.490,14.446,151.573
C03275=1103.064,117.100,-60.586,177.493,14.445,151.572
C03276=1103.070,117.350,-60.605,177.496,14.444,151.571
C03277=1103.075,117.598,-60.624,177.500,14.444,151.570
C03278=1103.080,117.848,-60.643,177.503,14.444,151.570
C03279=1103.086,118.097,-60.662,177.507,14.443,151.569
C03280=1103.092,118.347,-60.681,177.509,14.443,151.568
C03281=1103.098,118.596,-60.701,177.513,14.443,151.567
C03282=1103.103,118.845,-60.721,177.516,14.442,151.566
C03283=1103.109,119.094,-60.740,177.519,14.442,151.565
C03284=1103.114,119.343,-60.759,177.523,14.442,151.565
C03285=1103.120,119.592,-60.779,177.525,14.441,151.564
C03286=1103.126,119.841,-60.798,177.529,14.441,151.563
C03287=1103.132,120.091,-60.817,177.532,14.440,151.562
C03288=1103.137,120.340,-60.837,177.536,14.441,151.562
C03289=1103.143,120.588,-60.856,177.539,14.440,151.561
C03290=1103.148,120.838,-60.875,177.543,14.440,151.560
C03291=1103.153,121.088,-60.895,177.546,14.439,151.559
C03292=1103.159,121.337,-60.914,177.549,14.438,151.558
C03293=1103.165,121.586,-60.934,177.552,14.438,151.557
C03294=1103.171,121.835,-60.954,177.555,14.437,151.557
C03295=1103.176,122.085,-60.973,177.559,14.438,151.556
C03296=1103.182,122.334,-60.993,177.562,14.437,151.555
C03297=1103.187,122.582,-61.012,177.566,14.437,151.554
C03298=1103.193,122.831,-61.032,177.569,14.436,151.553
C03299=1103.199,123.080,-61.051,177.572,14.436,151.552
C03300=1103.205,123.330,-61.070,177.576,14.435,151.552
C03301=1103.210,123.579,-61.091,177.578,14.435,151.551
C03302=1103.216,123.828,-61.110,177.582,14.434,151.550
C03303=1103.222,124.077,-61.130,177.585,14.434,151.549
C03304=1103.227,124.327,-61.149,177.589,14.433,151.548
C03305=1103.233,124.576,-61.168,177.592,14.433,151.547
C03306=1103.239,124.825,-61.188,177.596,14.433,151.547
C03307=1103.245,125.074,-61.208,177.599,14.432,151.546
C03308=1103.250,125.324,-61.228,177.602,14.431,151.545
C03309=1103.256,125.573,-61.247,177.605,14.431,151.544
C03310=1103.262,125.822,-61.267,177.609,14.430,151.543
C03311=1103.267,126.071,-61.287,177.613,14.430,151.542
C03312=1103.273,126.320,-61.307,177.615,14.430,151.542
C03313=1103.279,126.569,-61.326,177.619,14.429,151.541
C03314=1103.284,126.819,-61.346,177.622,14.429,151.540
C03315=1103.290,127.068,-61.366,177.626,14.429,151.539
C03316=1103.296,127.317,-61.386,177.629,14.428,151.538
C03317=1103.302,127.566,-61.406,177.632,14.427,151.537
C03318=1103.308,127.838,-61.426,177.636,14.427,151.536
C03319=1103.314,128.110,-61.449,177.640,14.426,151.535
C03320=1103.320,128.383,-61.470,177.643,14.425,151.534
C03321=1103.327,128.655,-61.492,177.647,14.425,151.533
C03322=1103.333,128.904,-61.511,177.651,14.425,151.533
C03323=1103.338,129.154,-61.532,177.654,14.424,151.532
C03324=1103.344,129.402,-61.552,177.657,14.423,151.531
C03325=1103.350,129.652,-61.571,177.661,14.423,151.530
C03326=1103.356,129.901,-61.591,177.664,14.422,151.529
C03327=1103.361,130.150,-61.612,177.668,14.422,151.528
C03328=1103.367,130.399,-61.631,177.671,14.421,151.527
C03329=1103.373,130.648,-61.651,177.675,14.421,151.526
C03330=1103.379,130.897,-61.671,177.678,14.420,151.526
C03331=1103.384,131.147,-61.692,177.682,14.420,151.525
C03332=1103.390,131.396,-61.711,177.685,14.419,151.524
C03333=1103.396,131.645,-61.731,177.688,14.418,151.523
C03334=1103.401,131.894,-61.751,177.692,14.418,151.522
C03335=1103.407,132.143,-61.771,177.695,14.417,151.521
C03336=1103.413,132.392,-61.791,177.699,14.417,151.520
C03337=1103.418,132.641,-61.811,177.702,14.416,151.519
C03338=1103.424,132.890,-61.831,177.706,14.416,151.519
C03339=1103.430,133.139,-61.852,177.709,14.415,151.518
C03340=1103.435,133.389,-61.871,177.713,14.415,151.517
C03341=1103.441,133.638,-61.891,177.716,14.414,151.516
C03342=1103.447,133.887,-61.912,177.719,14.413,151.515
C03343=1103.453,134.136,-61.932,177.723,14.413,151.514
C03344=1103.458,134.385,-61.952,177.726,14.412,151.513
C03345=1103.464,134.634,-61.972,177.730,14.412,151.512
C03346=1103.470,134.883,-61.993,177.733,14.411,151.512
C03347=1103.475,135.133,-62.012,177.737,14.411,151.511
C03348=1103.480,135.382,-62.033,177.740,14.410,151.510
C03349=1103.486,135.631,-62.053,177.744,14.410,151.509
C03350=1103.492,135.880,-62.073,177.747,14.409,151.508
C03351=1103.498,136.129,-62.093,177.751,14.409,151.507
C03352=1103.504,136.378,-62.114,177.754,14.408,151.506
C03353=1103.510,136.627,-62.134,177.757,14.407,151.505
C03354=1103.515,136.876,-62.154,177.761,14.407,151.504
C03355=1103.521,137.125,-62.174,177.764,14.406,151.503
C03356=1103.526,137.374,-62.195,177.768,14.406,151.502
C03357=1103.532,137.623,-62.215,177.771,14.405,151.502
C03358=1103.538,137.873,-62.236,177.775,14.405,151.501
C03359=1103.544,138.122,-62.256,177.778,14.404,151.500
C03360=1103.549,138.371,-62.276,177.782,14.404,151.499
C03361=1103.554,138.620,-62.297,177.785,14.403,151.498
C03362=1103.560,138.869,-62.317,177.789,14.402,151.497
C03363=1103.566,139.119,-62.338,177.792,14.401,151.496
C03364=1103.572,139.367,-62.358,177.795,14.401,151.495
C03365=1103.578,139.617,-62.378,177.799,14.400,151.494
C03366=1103.583,139.866,-62.399,177.802,14.399,151.493
C03367=1103.589,140.114,-62.419,177.806,14.399,151.493
C03368=1103.595,140.364,-62.440,177.810,14.398,151.491
C03369=1103.601,140.613,-62.460,177.814,14.398,151.491
C03370=1103.606,140.862,-62.481,177.817,14.397,151.490
C03371=1103.611,141.111,-62.502,177.821,14.396,151.489
C03372=1103.617,141.360,-62.522,177.824,14.395,151.488
C03373=1103.623,141.609,-62.542,177.828,14.395,151.487
C03374=1103.629,141.858,-62.563,177.831,14.394,151.486
C03375=1103.634,142.108,-62.584,177.835,14.394,151.485
C03376=1103.640,142.356,-62.604,177.838,14.393,151.484
C03377=1103.646,142.606,-62.625,177.841,14.392,151.483
C03378=1103.651,142.855,-62.646,177.845,14.392,151.482
C03379=1103.657,143.104,-62.666,177.848,14.391,151.481
C03380=1103.662,143.353,-62.686,177.852,14.391,151.480
C03381=1103.668,143.601,-62.707,177.856,14.389,151.479
C03382=1103.674,143.874,-62.730,177.860,14.389,151.478
C03383=1103.680,144.146,-62.753,177.864,14.388,151.477
C03384=1103.686,144.419,-62.775,177.867,14.388,151.476
C03385=1103.694,144.691,-62.798,177.871,14.387,151.475
C03386=1103.699,144.940,-62.819,177.875,14.387,151.474
C03387=1103.704,145.189,-62.839,177.879,14.385,151.473
C03388=1103.710,145.437,-62.860,177.882,14.384,151.473
C03389=1103.716,145.687,-62.881,177.886,14.384,151.472
C03390=1103.722,145.936,-62.901,177.889,14.383,151.471
C03391=1103.727,146.185,-62.923,177.893,14.383,151.470
C03392=1103.733,146.434,-62.943,177.896,14.382,151.469
C03393=1103.738,146.684,-62.964,177.900,14.381,151.468
C03394=1103.744,146.932,-62.985,177.904,14.380,151.467
C03395=1103.750,147.182,-63.006,177.907,14.380,151.466
C03396=1103.756,147.431,-63.026,177.911,14.379,151.465
C03397=1103.761,147.679,-63.047,177.915,14.379,151.464
C03398=1103.767,147.929,-63.068,177.918,14.378,151.463
C03399=1103.773,148.178,-63.090,177.922,14.377,151.462
C03400=1103.778,148.427,-63.110,177.925,14.376,151.461
C03401=1103.785,148.676,-63.131,177.929,14.375,151.460
C03402=1103.790,148.925,-63.152,177.933,14.375,151.459
C03403=1103.796,149.173,-63.173,177.936,14.374,151.458
C03404=1103.801,149.423,-63.194,177.940,14.373,151.457
C03405=1103.807,149.671,-63.215,177.943,14.372,151.456
C03406=1103.813,149.921,-63.236,177.947,14.372,151.455
C03407=1103.818,150.170,-63.257,177.951,14.371,151.454
C03408=1103.824,150.419,-63.278,177.955,14.370,151.453
C03409=1103.830,150.668,-63.300,177.958,14.369,151.452
C03410=1103.835,150.917,-63.320,177.962,14.369,151.451
C03411=1103.841,151.166,-63.341,177.965,14.368,151.450
C03412=1103.847,151.416,-63.362,177.969,14.368,151.449
C03413=1103.852,151.664,-63.384,177.972,14.367,151.449
C03414=1103.858,151.914,-63.405,177.977,14.366,151.447
C03415=1103.863,152.162,-63.426,177.980,14.365,151.447
C03416=1103.869,152.411,-63.447,177.984,14.364,151.445
C03417=1103.875,152.661,-63.468,177.987,14.364,151.445
C03418=1103.880,152.909,-63.489,177.991,14.362,151.443
C03419=1103.887,153.158,-63.511,177.995,14.362,151.443
C03420=1103.892,153.408,-63.531,177.998,14.361,151.442
C03421=1103.897,153.656,-63.553,178.002,14.360,151.441
C03422=1103.904,153.905,-63.574,178.005,14.360,151.440
C03423=1103.909,154.154,-63.595,178.009,14.359,151.439
C03424=1103.914,154.404,-63.617,178.013,14.358,151.438
C03425=1103.920,154.652,-63.638,178.017,14.357,151.437
C03426=1103.926,154.902,-63.659,178.020,14.356,151.436
C03427=1103.931,155.151,-63.681,178.024,14.356,151.435
C03428=1103.937,155.400,-63.702,178.027,14.355,151.434
C03429=1103.943,155.649,-63.724,178.032,14.354,151.433
C03430=1103.949,155.898,-63.744,178.035,14.353,151.432
C03431=1103.954,156.147,-63.766,178.039,14.353,151.431
C03432=1103.961,156.396,-63.787,178.043,14.351,151.430
C03433=1103.965,156.645,-63.809,178.047,14.351,151.429
C03434=1103.972,156.894,-63.831,178.050,14.350,151.428
C03435=1103.977,157.143,-63.851,178.053,14.349,151.427
C03436=1103.982,157.392,-63.873,178.057,14.348,151.426
C03437=1103.989,157.641,-63.894,178.061,14.347,151.425
C03438=1103.994,157.889,-63.916,178.065,14.347,151.424
C03439=1104.000,158.139,-63.938,178.068,14.345,151.422
C03440=1104.006,158.388,-63.959,178.072,14.345,151.422
C03441=1104.011,158.637,-63.980,178.076,14.344,151.420
C03442=1104.017,158.886,-64.002,178.080,14.344,151.420
C03443=1104.022,159.135,-64.024,178.083,14.342,151.419
C03444=1104.028,159.384,-64.045,178.087,14.342,151.417
C03445=1104.034,159.633,-64.066,178.091,14.341,151.417
C03446=1104.040,159.905,-64.090,178.095,14.340,151.415
C03447=1104.046,160.177,-64.114,178.099,14.339,151.414
C03448=1104.053,160.449,-64.138,178.103,14.338,151.413
C03449=1104.059,160.721,-64.161,178.107,14.337,151.412
C03450=1104.065,160.969,-64.182,178.111,14.336,151.411
C03451=1104.070,161.219,-64.205,178.115,14.335,151.410
C03452=1104.076,161.468,-64.226,178.118,14.334,151.409
C03453=1104.082,161.716,-64.247,178.122,14.334,151.408
C03454=1104.087,161.966,-64.270,178.126,14.332,151.407
C03455=1104.093,162.214,-64.291,178.130,14.332,151.406
C03456=1104.098,162.464,-64.313,178.133,14.331,151.405
C03457=1104.104,162.712,-64.334,178.137,14.330,151.404
C03458=1104.109,162.962,-64.357,178.141,14.329,151.403
C03459=1104.115,163.210,-64.378,178.145,14.329,151.402
C03460=1104.120,163.460,-64.400,178.148,14.327,151.401
C03461=1104.126,163.708,-64.421,178.152,14.327,151.400
C03462=1104.132,163.958,-64.443,178.156,14.326,151.399
C03463=1104.137,164.207,-64.465,178.160,14.325,151.398
C03464=1104.143,164.456,-64.487,178.163,14.324,151.397
C03465=1104.149,164.705,-64.510,178.167,14.324,151.396
C03466=1104.154,164.953,-64.531,178.171,14.322,151.395
C03467=1104.159,165.203,-64.553,178.175,14.322,151.393
C03468=1104.164,165.451,-64.575,178.179,14.320,151.392
C03469=1104.170,165.701,-64.597,178.183,14.320,151.391
C03470=1104.176,165.950,-64.619,178.186,14.319,151.390
C03471=1104.182,166.198,-64.641,178.190,14.318,151.389
C03472=1104.187,166.448,-64.663,178.194,14.317,151.388
C03473=1104.193,166.696,-64.684,178.198,14.316,151.387
C03474=1104.198,166.946,-64.706,178.201,14.316,151.386
C03475=1104.205,167.194,-64.729,178.205,14.315,151.385
C03476=1104.209,167.443,-64.751,178.209,14.314,151.384
C03477=1104.216,167.692,-64.772,178.213,14.313,151.383
C03478=1104.221,167.942,-64.795,178.217,14.312,151.382
C03479=1104.226,168.190,-64.817,178.221,14.311,151.381
C03480=1104.232,168.439,-64.839,178.224,14.310,151.380
C03481=1104.238,168.689,-64.861,178.228,14.310,151.379
C03482=1104.244,168.936,-64.883,178.232,14.308,151.378
C03483=1104.249,169.186,-64.905,178.236,14.308,151.377
C03484=1104.254,169.436,-64.927,178.240,14.306,151.376
C03485=1104.260,169.683,-64.949,178.244,14.306,151.375
C03486=1104.266,169.933,-64.972,178.247,14.304,151.374
C03487=1104.272,170.182,-64.993,178.252,14.304,151.372
C03488=1104.277,170.430,-65.016,178.255,14.303,151.371
C03489=1104.283,170.680,-65.038,178.259,14.302,151.370
C03490=1104.289,170.928,-65.060,178.263,14.301,151.369
C03491=1104.294,171.178,-65.083,178.266,14.299,151.368
C03492=1104.299,171.427,-65.105,178.271,14.299,151.367
C03493=1104.306,171.675,-65.127,178.274,14.297,151.366
C03494=1104.311,171.925,-65.149,178.278,14.297,151.365
C03495=1104.317,172.174,-65.172,178.282,14.296,151.364
C03496=1104.322,172.422,-65.193,178.286,14.295,151.363
C03497=1104.328,172.671,-65.216,178.289,14.294,151.362
C03498=1104.334,172.921,-65.239,178.294,14.293,151.361
C03499=1104.340,173.169,-65.261,178.297,14.292,151.360
C03500=1104.345,173.418,-65.283,178.301,14.291,151.358
C03501=1104.351,173.667,-65.306,178.305,14.290,151.357
C03502=1104.357,173.916,-65.328,178.309,14.289,151.356
C03503=1104.362,174.165,-65.350,178.313,14.288,151.355
C03504=1104.368,174.414,-65.373,178.317,14.287,151.354
C03505=1104.374,174.662,-65.394,178.321,14.286,151.353
C03506=1104.380,174.911,-65.417,178.325,14.285,151.352
C03507=1104.385,175.161,-65.440,178.329,14.284,151.351
C03508=1104.391,175.410,-65.463,178.333,14.283,151.350
C03509=1104.397,175.658,-65.485,178.336,14.282,151.349
C03510=1104.403,175.930,-65.510,178.341,14.281,151.347
C03511=1104.409,176.202,-65.534,178.345,14.280,151.346
C03512=1104.415,176.473,-65.559,178.349,14.278,151.345
C03513=1104.422,176.745,-65.583,178.354,14.278,151.344
C03514=1104.428,176.994,-65.606,178.358,14.277,151.343
C03515=1104.433,177.242,-65.628,178.362,14.275,151.341
C03516=1104.438,177.491,-65.651,178.366,14.275,151.340
C03517=1104.445,177.740,-65.673,178.369,14.273,151.339
C03518=1104.450,177.989,-65.696,178.374,14.272,151.338
C03519=1104.456,178.238,-65.719,178.377,14.271,151.337
C03520=1104.462,178.487,-65.741,178.381,14.270,151.336
C03521=1104.467,178.736,-65.764,178.385,14.269,151.335
C03522=1104.473,178.985,-65.787,178.389,14.268,151.334
C03523=1104.479,179.234,-65.809,178.393,14.267,151.333
C03524=1104.485,179.483,-65.832,178.397,14.266,151.331
C03525=1104.490,179.731,-65.854,178.401,14.265,151.330
C03526=1104.496,179.980,-65.877,178.405,14.263,151.329
C03527=1104.501,180.229,-65.900,178.409,14.263,151.328
C03528=1104.507,180.478,-65.923,178.413,14.261,151.327
C03529=1104.514,180.727,-65.945,178.417,14.260,151.326
C03530=1104.519,180.976,-65.968,178.421,14.259,151.325
C03531=1104.525,181.224,-65.991,178.425,14.258,151.323
C03532=1104.531,181.474,-66.014,178.429,14.257,151.322
C03533=1104.536,181.723,-66.036,178.433,14.256,151.321
C03534=1104.542,181.972,-66.059,178.437,14.255,151.320
C03535=1104.548,182.221,-66.082,178.441,14.254,151.319
C03536=1104.553,182.470,-66.105,178.445,14.252,151.318
C03537=1104.560,182.718,-66.128,178.449,14.252,151.317
C03538=1104.566,182.967,-66.151,178.453,14.250,151.315
C03539=1104.571,183.216,-66.174,178.457,14.250,151.314
C03540=1104.577,183.465,-66.196,178.461,14.248,151.313
C03541=1104.583,183.714,-66.219,178.465,14.247,151.312
C03542=1104.589,183.963,-66.242,178.469,14.246,151.311
C03543=1104.594,184.211,-66.265,178.473,14.245,151.310
C03544=1104.600,184.460,-66.288,178.477,14.244,151.309
C03545=1104.606,184.709,-66.311,178.481,14.243,151.307
C03546=1104.612,184.958,-66.334,178.485,14.242,151.306
C03547=1104.618,185.206,-66.358,178.489,14.240,151.305
C03548=1104.623,185.455,-66.381,178.493,14.239,151.304
C03549=1104.629,185.704,-66.404,178.498,14.238,151.303
C03550=1104.635,185.953,-66.427,178.501,14.237,151.302
C03551=1104.640,186.202,-66.450,178.505,14.236,151.301
C03552=1104.645,186.451,-66.473,178.509,14.235,151.299
C03553=1104.651,186.700,-66.496,178.513,14.234,151.298
C03554=1104.657,186.949,-66.519,178.517,14.232,151.297
C03555=1104.663,187.198,-66.542,178.521,14.232,151.296
C03556=1104.668,187.447,-66.566,178.525,14.231,151.295
C03557=1104.674,187.695,-66.589,178.529,14.230,151.294
C03558=1104.679,187.944,-66.612,178.533,14.228,151.293
C03559=1104.685,188.193,-66.635,178.538,14.227,151.291
C03560=1104.690,188.442,-66.659,178.541,14.226,151.290
C03561=1104.696,188.691,-66.682,178.546,14.225,151.289
C03562=1104.702,188.940,-66.705,178.549,14.224,151.288
C03563=1104.708,189.188,-66.728,178.554,14.223,151.287
C03564=1104.713,189.438,-66.752,178.557,14.222,151.286
C03565=1104.719,189.686,-66.775,178.562,14.221,151.284
C03566=1104.724,189.935,-66.798,178.565,14.220,151.283
C03567=1104.730,190.184,-66.821,178.570,14.219,151.282
C03568=1104.735,190.433,-66.845,178.573,14.217,151.281
C03569=1104.741,190.681,-66.868,178.578,14.216,151.280
C03570=1104.748,190.931,-66.892,178.581,14.215,151.279
C03571=1104.753,191.180,-66.915,178.586,14.214,151.277
C03572=1104.759,191.428,-66.939,178.590,14.213,151.276
C03573=1104.764,191.677,-66.962,178.594,14.212,151.275
C03574=1104.771,191.948,-66.987,178.598,14.210,151.274
C03575=1104.776,192.220,-67.013,178.603,14.209,151.273
C03576=1104.782,192.491,-67.039,178.607,14.208,151.271
C03577=1104.789,192.762,-67.064,178.612,14.207,151.270
C03578=1104.794,193.010,-67.088,178.615,14.206,151.269
C03579=1104.800,193.259,-67.111,178.620,14.205,151.268
C03580=1104.806,193.508,-67.135,178.624,14.203,151.266
C03581=1104.811,193.757,-67.159,178.628,14.202,151.265
C03582=1104.817,194.006,-67.182,178.632,14.201,151.264
C03583=1104.823,194.255,-67.205,178.637,14.200,151.263
C03584=1104.828,194.504,-67.229,178.640,14.199,151.262
C03585=1104.834,194.752,-67.253,178.645,14.198,151.261
C03586=1104.840,195.001,-67.277,178.648,14.196,151.259
C03587=1104.846,195.250,-67.300,178.653,14.195,151.258
C03588=1104.852,195.499,-67.324,178.657,14.194,151.257
C03589=1104.857,195.748,-67.347,178.661,14.193,151.256
C03590=1104.863,195.996,-67.371,178.665,14.191,151.255
C03591=1104.868,196.245,-67.394,178.669,14.191,151.254
C03592=1104.875,196.494,-67.419,178.673,14.189,151.252
C03593=1104.880,196.743,-67.442,178.678,14.188,151.251
C03594=1104.886,196.992,-67.466,178.681,14.186,151.250
C03595=1104.892,197.240,-67.489,178.686,14.186,151.249
C03596=1104.897,197.489,-67.513,178.690,14.184,151.247
C03597=1104.903,197.738,-67.537,178.694,14.183,151.246
C03598=1104.909,197.987,-67.561,178.698,14.182,151.245
C03599=1104.914,198.236,-67.584,178.703,14.181,151.244
C03600=1104.920,198.484,-67.608,178.706,14.179,151.243
C03601=1104.926,198.733,-67.632,178.711,14.178,151.241
C03602=1104.931,198.982,-67.656,178.714,14.177,151.240
C03603=1104.937,199.231,-67.680,178.719,14.176,151.239
C03604=1104.943,199.480,-67.704,178.723,14.174,151.238
C03605=1104.949,199.728,-67.728,178.727,14.173,151.237
C03606=1104.954,199.977,-67.751,178.731,14.172,151.235
C03607=1104.960,200.226,-67.775,178.736,14.171,151.234
C03608=1104.966,200.475,-67.800,178.739,14.169,151.233
C03609=1104.972,200.723,-67.823,178.744,14.168,151.232
C03610=1104.977,200.972,-67.848,178.748,14.167,151.230
C03611=1104.984,201.222,-67.871,178.752,14.166,151.229
C03612=1104.989,201.470,-67.895,178.756,14.164,151.228
C03613=1104.995,201.718,-67.919,178.761,14.163,151.227
C03614=1105.001,201.968,-67.944,178.765,14.162,151.226
C03615=1105.006,202.216,-67.968,178.769,14.161,151.224
C03616=1105.012,202.465,-67.991,178.773,14.159,151.223
C03617=1105.018,202.714,-68.016,178.778,14.158,151.222
C03618=1105.024,202.962,-68.040,178.781,14.156,151.221
C03619=1105.029,203.211,-68.063,178.786,14.156,151.219
C03620=1105.035,203.461,-68.088,178.789,14.154,151.218
C03621=1105.041,203.709,-68.112,178.794,14.153,151.217
C03622=1105.047,203.957,-68.136,178.798,14.152,151.216
C03623=1105.052,204.207,-68.160,178.802,14.151,151.215
C03624=1105.058,204.455,-68.185,178.806,14.149,151.213
C03625=1105.064,204.704,-68.208,178.811,14.148,151.212
C03626=1105.070,204.953,-68.233,178.815,14.147,151.211
C03627=1105.075,205.201,-68.257,178.819,14.146,151.210
